LIN {X 0,Y 332.118,Z 721.88,A -85,B 0,C 180,E1 -12190.22,E2 -12190.22} C_VEL
LIN {X 0,Y 333.86,Z 711.932,A -85,B 0,C 180,E1 -12192.438,E2 -12192.438} C_VEL
LIN {X 0,Y 335.853,Z 699.998,A -85,B 0,C 180,E1 -12194.532,E2 -12194.532} C_VEL
LIN {X 0,Y 337.763,Z 687.766,A -85,B 0,C 180,E1 -12196.241,E2 -12196.241} C_VEL
LIN {X 0,Y 339.691,Z 673.523,A -85,B 0,C 180,E1 -12197.797,E2 -12197.797} C_VEL
LIN {X 0,Y 341.315,Z 659.406,A -85,B 0,C 180,E1 -12198.989,E2 -12198.989} C_VEL
LIN {X 0,Y 342.676,Z 643.422,A -85,B 0,C 180,E1 -12199.976,E2 -12199.976} C_VEL
LIN {X 0,Y 343.599,Z 627.214,A -85,B 0,C 180,E1 -12200.656,E2 -12200.656} C_VEL
LIN {X 0,Y 345.215,Z 570.987,A -85,B 0,C 180,E1 -12201.908,E2 -12201.908} C_VEL
LIN {X 0,Y 347.175,Z 499.948,A -85,B 0,C 180,E1 -12203.441,E2 -12203.441} C_VEL
LIN {X 0,Y 345.23,Z 482.09,A -85,B 0,C 180,E1 -12204.102,E2 -12204.102} C_VEL
LIN {X 0,Y 348.72,Z 438.304,A -85,B 0,C 180,E1 -12208.447,E2 -12208.447} C_VEL
LIN {X 0,Y 351.971,Z 398.894,A -85,B 0,C 180,E1 -12212.333,E2 -12212.333} C_VEL
LIN {X 0,Y 355.002,Z 360.835,A -85,B 0,C 180,E1 -12216.072,E2 -12216.072} C_VEL
LIN {X 0,Y 355.314,Z 355.414,A -85,B 0,C 180,E1 -12216.623,E2 -12216.623} C_VEL
LIN {X 0,Y 350.277,Z 339.623,A -85,B 0,C 180,E1 -12219.095,E2 -12219.095} C_VEL
LIN {X 0,Y 344.773,Z 325.615,A -85,B 0,C 180,E1 -12221.572,E2 -12221.572} C_VEL
LIN {X 0,Y 338.807,Z 312.634,A -85,B 0,C 180,E1 -12224.158,E2 -12224.158} C_VEL
LIN {X 0,Y 334.604,Z 304.41,A -85,B 0,C 180,E1 -12225.992,E2 -12225.992} C_VEL
LIN {X 0,Y 332,Z 299.711,A -85,B 0,C 180,E1 -12227.122,E2 -12227.122} C_VEL
LIN {X 0,Y 330.195,Z 296.3,A -85,B 0,C 180,E1 -12227.959,E2 -12227.959} C_VEL
LIN {X 0,Y 330.046,Z 295.41,A -85,B 0,C 180,E1 -12228.363,E2 -12228.363} C_VEL
LIN {X 0,Y 330.062,Z 295.372,A -85,B 0,C 180,E1 -12232.69,E2 -12232.69} C_VEL
LIN {X 0,Y 330.038,Z 295.376,A -85,B 0,C 180,E1 -12237.047,E2 -12237.047} C_VEL
LIN {X 0,Y 330.027,Z 295.369,A -85,B 0,C 180,E1 -12241.388,E2 -12241.388} C_VEL
LIN {X 0,Y 330.023,Z 295.376,A -85,B 0,C 180,E1 -12245.737,E2 -12245.737} C_VEL
LIN {X 0,Y 330.026,Z 295.368,A -85,B 0,C 180,E1 -12250.12,E2 -12250.12} C_VEL
LIN {X 0,Y 330.038,Z 295.376,A -85,B 0,C 180,E1 -12254.383,E2 -12254.383} C_VEL
LIN {X 0,Y 330.048,Z 295.365,A -85,B 0,C 180,E1 -12258.73,E2 -12258.73} C_VEL
LIN {X 0,Y 330.059,Z 295.37,A -85,B 0,C 180,E1 -12263.003,E2 -12263.003} C_VEL
LIN {X 0,Y 330.042,Z 295.369,A -85,B 0,C 180,E1 -12267.427,E2 -12267.427} C_VEL
LIN {X 0,Y 330.036,Z 295.371,A -85,B 0,C 180,E1 -12271.651,E2 -12271.651} C_VEL
LIN {X 0,Y 330.069,Z 295.642,A -85,B 0,C 180,E1 -12274.026,E2 -12274.026} C_VEL
LIN {X 0,Y 331.671,Z 299.336,A -85,B 0,C 180,E1 -12274.943,E2 -12274.943} C_VEL
LIN {X 0,Y 339.158,Z 316.344,A -85,B 0,C 180,E1 -12278.681,E2 -12278.681} C_VEL
LIN {X 0,Y 341.505,Z 321.378,A -85,B 0,C 180,E1 -12279.662,E2 -12279.662} C_VEL
LIN {X 0,Y 357.451,Z 348.34,A -85,B 0,C 180,E1 -12282.794,E2 -12282.794} C_VEL
LIN {X 0,Y 370.048,Z 371.248,A -85,B 0,C 180,E1 -12285.081,E2 -12285.081} C_VEL
LIN {X 0,Y 357.996,Z 576.955,A -85,B 0,C 180,E1 -12290.185,E2 -12290.185} C_VEL
LIN {X 0,Y 355.992,Z 598.538,A -85,B 0,C 180,E1 -12291.003,E2 -12291.003} C_VEL
LIN {X 0,Y 353.569,Z 618.824,A -85,B 0,C 180,E1 -12292.056,E2 -12292.056} C_VEL
LIN {X 0,Y 350.696,Z 639.126,A -85,B 0,C 180,E1 -12293.428,E2 -12293.428} C_VEL
LIN {X 0,Y 347.572,Z 658.567,A -85,B 0,C 180,E1 -12295.081,E2 -12295.081} C_VEL
LIN {X 0,Y 344.166,Z 677.781,A -85,B 0,C 180,E1 -12297.096,E2 -12297.096} C_VEL
LIN {X 0,Y 340.909,Z 695.134,A -85,B 0,C 180,E1 -12299.317,E2 -12299.317} C_VEL
LIN {X 0,Y 337.768,Z 711.391,A -85,B 0,C 180,E1 -12301.829,E2 -12301.829} C_VEL
LIN {X 0,Y 334.968,Z 725.97,A -85,B 0,C 180,E1 -12304.546,E2 -12304.546} C_VEL
LIN {X 0,Y 332.525,Z 739.34,A -85,B 0,C 180,E1 -12307.553,E2 -12307.553} C_VEL
LIN {X 0,Y 330.674,Z 750.572,A -85,B 0,C 180,E1 -12310.628,E2 -12310.628} C_VEL
LIN {X 0,Y 329.371,Z 759.964,A -85,B 0,C 180,E1 -12313.785,E2 -12313.785} C_VEL
LIN {X 0,Y 328.56,Z 767.582,A -85,B 0,C 180,E1 -12316.988,E2 -12316.988} C_VEL
LIN {X 0,Y 328.163,Z 773.719,A -85,B 0,C 180,E1 -12320.355,E2 -12320.355} C_VEL
LIN {X 0,Y 328.074,Z 777.864,A -85,B 0,C 180,E1 -12323.527,E2 -12323.527} C_VEL
LIN {X 0,Y 328.085,Z 780.383,A -85,B 0,C 180,E1 -12326.682,E2 -12326.682} C_VEL
LIN {X 0,Y 328.118,Z 781.355,A -85,B 0,C 180,E1 -12329.827,E2 -12329.827} C_VEL
LIN {X 0,Y 328.075,Z 780.859,A -85,B 0,C 180,E1 -12332.972,E2 -12332.972} C_VEL
LIN {X 0,Y 328.045,Z 778.829,A -85,B 0,C 180,E1 -12336.126,E2 -12336.126} C_VEL
LIN {X 0,Y 328.116,Z 775.251,A -85,B 0,C 180,E1 -12339.296,E2 -12339.296} C_VEL
LIN {X 0,Y 328.493,Z 769.816,A -85,B 0,C 180,E1 -12342.661,E2 -12342.661} C_VEL
LIN {X 0,Y 329.298,Z 763.002,A -85,B 0,C 180,E1 -12345.861,E2 -12345.861} C_VEL
LIN {X 0,Y 330.734,Z 753.863,A -85,B 0,C 180,E1 -12349.242,E2 -12349.242} C_VEL
LIN {X 0,Y 332.904,Z 742.52,A -85,B 0,C 180,E1 -12352.611,E2 -12352.611} C_VEL
LIN {X 0,Y 335.725,Z 729.474,A -85,B 0,C 180,E1 -12355.775,E2 -12355.775} C_VEL
LIN {X 0,Y 339.122,Z 714.749,A -85,B 0,C 180,E1 -12358.725,E2 -12358.725} C_VEL
LIN {X 0,Y 343.041,Z 698.333,A -85,B 0,C 180,E1 -12361.45,E2 -12361.45} C_VEL
LIN {X 0,Y 347.215,Z 680.841,A -85,B 0,C 180,E1 -12363.865,E2 -12363.865} C_VEL
LIN {X 0,Y 351.726,Z 661.714,A -85,B 0,C 180,E1 -12366.048,E2 -12366.048} C_VEL
LIN {X 0,Y 356.386,Z 641.227,A -85,B 0,C 180,E1 -12367.968,E2 -12367.968} C_VEL
LIN {X 0,Y 360.995,Z 620.134,A -85,B 0,C 180,E1 -12369.573,E2 -12369.573} C_VEL
LIN {X 0,Y 365.603,Z 597.763,A -85,B 0,C 180,E1 -12370.92,E2 -12370.92} C_VEL
LIN {X 0,Y 370.108,Z 573.956,A -85,B 0,C 180,E1 -12372.002,E2 -12372.002} C_VEL
LIN {X 0,Y 380.25,Z 515.563,A -85,B 0,C 180,E1 -12374.095,E2 -12374.095} C_VEL
LIN {X 0,Y 391.481,Z 464.537,A -85,B 0,C 180,E1 -12375.931,E2 -12375.931} C_VEL
LIN {X 0,Y 399.695,Z 432.421,A -85,B 0,C 180,E1 -12377.075,E2 -12377.075} C_VEL
LIN {X 0,Y 383.918,Z 497.009,A -85,B 0,C 180,E1 -12379.426,E2 -12379.426} C_VEL
LIN {X 0,Y 372.15,Z 555.463,A -85,B 0,C 180,E1 -12381.651,E2 -12381.651} C_VEL
LIN {X 0,Y 367.645,Z 579.27,A -85,B 0,C 180,E1 -12382.665,E2 -12382.665} C_VEL
LIN {X 0,Y 363.116,Z 600.549,A -85,B 0,C 180,E1 -12383.896,E2 -12383.896} C_VEL
LIN {X 0,Y 358.234,Z 621.939,A -85,B 0,C 180,E1 -12385.488,E2 -12385.488} C_VEL
LIN {X 0,Y 353.563,Z 641.476,A -85,B 0,C 180,E1 -12387.308,E2 -12387.308} C_VEL
LIN {X 0,Y 349.098,Z 659.317,A -85,B 0,C 180,E1 -12389.349,E2 -12389.349} C_VEL
LIN {X 0,Y 344.901,Z 675.585,A -85,B 0,C 180,E1 -12391.613,E2 -12391.613} C_VEL
LIN {X 0,Y 341.034,Z 690.337,A -85,B 0,C 180,E1 -12394.098,E2 -12394.098} C_VEL
LIN {X 0,Y 337.575,Z 703.545,A -85,B 0,C 180,E1 -12396.801,E2 -12396.801} C_VEL
LIN {X 0,Y 334.599,Z 715.171,A -85,B 0,C 180,E1 -12399.719,E2 -12399.719} C_VEL
LIN {X 0,Y 332.292,Z 724.649,A -85,B 0,C 180,E1 -12402.67,E2 -12402.67} C_VEL
LIN {X 0,Y 330.597,Z 732.231,A -85,B 0,C 180,E1 -12405.641,E2 -12405.641} C_VEL
LIN {X 0,Y 329.386,Z 738.403,A -85,B 0,C 180,E1 -12408.798,E2 -12408.798} C_VEL
LIN {X 0,Y 328.658,Z 742.803,A -85,B 0,C 180,E1 -12411.956,E2 -12411.956} C_VEL
LIN {X 0,Y 328.278,Z 745.629,A -85,B 0,C 180,E1 -12415.284,E2 -12415.284} C_VEL
LIN {X 0,Y 328.142,Z 746.633,A -85,B 0,C 180,E1 -12418.429,E2 -12418.429} C_VEL
LIN {X 0,Y 328.103,Z 746.012,A -85,B 0,C 180,E1 -12421.572,E2 -12421.572} C_VEL
LIN {X 0,Y 328.151,Z 743.758,A -85,B 0,C 180,E1 -12424.72,E2 -12424.72} C_VEL
LIN {X 0,Y 328.372,Z 739.807,A -85,B 0,C 180,E1 -12427.876,E2 -12427.876} C_VEL
LIN {X 0,Y 328.849,Z 734.444,A -85,B 0,C 180,E1 -12430.867,E2 -12430.867} C_VEL
LIN {X 0,Y 329.72,Z 727.043,A -85,B 0,C 180,E1 -12433.975,E2 -12433.975} C_VEL
LIN {X 0,Y 330.982,Z 718.343,A -85,B 0,C 180,E1 -12436.859,E2 -12436.859} C_VEL
LIN {X 0,Y 332.702,Z 707.869,A -85,B 0,C 180,E1 -12439.67,E2 -12439.67} C_VEL
LIN {X 0,Y 334.795,Z 695.999,A -85,B 0,C 180,E1 -12442.29,E2 -12442.29} C_VEL
LIN {X 0,Y 337.291,Z 682.225,A -85,B 0,C 180,E1 -12444.801,E2 -12444.801} C_VEL
LIN {X 0,Y 339.946,Z 667.484,A -85,B 0,C 180,E1 -12447.028,E2 -12447.028} C_VEL
LIN {X 0,Y 342.754,Z 651.22,A -85,B 0,C 180,E1 -12449.059,E2 -12449.059} C_VEL
LIN {X 0,Y 345.512,Z 634.102,A -85,B 0,C 180,E1 -12450.812,E2 -12450.812} C_VEL
LIN {X 0,Y 348.253,Z 615.141,A -85,B 0,C 180,E1 -12452.376,E2 -12452.376} C_VEL
LIN {X 0,Y 350.723,Z 595.391,A -85,B 0,C 180,E1 -12453.647,E2 -12453.647} C_VEL
LIN {X 0,Y 352.768,Z 575.246,A -85,B 0,C 180,E1 -12454.618,E2 -12454.618} C_VEL
LIN {X 0,Y 354.34,Z 554.645,A -85,B 0,C 180,E1 -12455.306,E2 -12455.306} C_VEL
LIN {X 0,Y 364.432,Z 383.187,A -85,B 0,C 180,E1 -12459.733,E2 -12459.733} C_VEL
LIN {X 0,Y 362.119,Z 366.133,A -85,B 0,C 180,E1 -12460.564,E2 -12460.564} C_VEL
LIN {X 0,Y 348.934,Z 341.464,A -85,B 0,C 180,E1 -12463.054,E2 -12463.054} C_VEL
LIN {X 0,Y 347.117,Z 337.74,A -85,B 0,C 180,E1 -12463.507,E2 -12463.507} C_VEL
LIN {X 0,Y 339.998,Z 319.459,A -85,B 0,C 180,E1 -12467.208,E2 -12467.208} C_VEL
LIN {X 0,Y 333.092,Z 302.809,A -85,B 0,C 180,E1 -12470.921,E2 -12470.921} C_VEL
LIN {X 0,Y 330.076,Z 295.57,A -85,B 0,C 180,E1 -12472.715,E2 -12472.715} C_VEL
LIN {X 0,Y 330.043,Z 295.371,A -85,B 0,C 180,E1 -12477.054,E2 -12477.054} C_VEL
LIN {X 0,Y 330.044,Z 295.349,A -85,B 0,C 180,E1 -12481.469,E2 -12481.469} C_VEL
LIN {X 0,Y 330.072,Z 295.561,A -85,B 0,C 180,E1 -12483.653,E2 -12483.653} C_VEL
LIN {X 0,Y 330.669,Z 297.596,A -85,B 0,C 180,E1 -12484.103,E2 -12484.103} C_VEL
LIN {X 0,Y 332.502,Z 301.305,A -85,B 0,C 180,E1 -12484.843,E2 -12484.843} C_VEL
LIN {X 0,Y 338.631,Z 314.413,A -85,B 0,C 180,E1 -12487.335,E2 -12487.335} C_VEL
LIN {X 0,Y 346.07,Z 332.865,A -85,B 0,C 180,E1 -12490.496,E2 -12490.496} C_VEL
LIN {X 0,Y 352.203,Z 350.651,A -85,B 0,C 180,E1 -12493.251,E2 -12493.251} C_VEL
LIN {X 0,Y 353.624,Z 356.013,A -85,B 0,C 180,E1 -12494.018,E2 -12494.018} C_VEL
LIN {X 0,Y 350.25,Z 397.698,A -85,B 0,C 180,E1 -12498.188,E2 -12498.188} C_VEL
LIN {X 0,Y 346.855,Z 438.589,A -85,B 0,C 180,E1 -12502.295,E2 -12502.295} C_VEL
LIN {X 0,Y 343.61,Z 481.813,A -85,B 0,C 180,E1 -12506.589,E2 -12506.589} C_VEL
LIN {X 0,Y 345.615,Z 502.467,A -85,B 0,C 180,E1 -12507.247,E2 -12507.247} C_VEL
LIN {X 0,Y 344.007,Z 560.903,A -85,B 0,C 180,E1 -12508.478,E2 -12508.478} C_VEL
LIN {X 0,Y 342.903,Z 568.569,A -85,B 0,C 180,E1 -12508.569,E2 -12508.569} C_VEL
LIN {X 0,Y 336.694,Z 588.888,A -85,B 0,C 180,E1 -12508.554,E2 -12508.554} C_VEL
LIN {X 0,Y 335.813,Z 595.472,A -85,B 0,C 180,E1 -12508.639,E2 -12508.639} C_VEL
LIN {X 0,Y 334.887,Z 627.398,A -85,B 0,C 180,E1 -12509.389,E2 -12509.389} C_VEL
LIN {X 0,Y 333.893,Z 644.369,A -85,B 0,C 180,E1 -12510.132,E2 -12510.132} C_VEL
LIN {X 0,Y 332.58,Z 659.659,A -85,B 0,C 180,E1 -12511.118,E2 -12511.118} C_VEL
LIN {X 0,Y 330.794,Z 675.437,A -85,B 0,C 180,E1 -12512.51,E2 -12512.51} C_VEL
LIN {X 0,Y 328.935,Z 689.154,A -85,B 0,C 180,E1 -12514.094,E2 -12514.094} C_VEL
LIN {X 0,Y 326.922,Z 702.47,A -85,B 0,C 180,E1 -12516.055,E2 -12516.055} C_VEL
LIN {X 0,Y 325.117,Z 713.568,A -85,B 0,C 180,E1 -12518.131,E2 -12518.131} C_VEL
LIN {X 0,Y 323.428,Z 723.844,A -85,B 0,C 180,E1 -12520.551,E2 -12520.551} C_VEL
LIN {X 0,Y 322.094,Z 732.194,A -85,B 0,C 180,E1 -12523.095,E2 -12523.095} C_VEL
LIN {X 0,Y 321.1,Z 739.181,A -85,B 0,C 180,E1 -12525.901,E2 -12525.901} C_VEL
LIN {X 0,Y 320.51,Z 744.121,A -85,B 0,C 180,E1 -12528.74,E2 -12528.74} C_VEL
LIN {X 0,Y 320.237,Z 747.308,A -85,B 0,C 180,E1 -12531.616,E2 -12531.616} C_VEL
LIN {X 0,Y 320.153,Z 748.689,A -85,B 0,C 180,E1 -12534.54,E2 -12534.54} C_VEL
LIN {X 0,Y 320.208,Z 748.308,A -85,B 0,C 180,E1 -12537.525,E2 -12537.525} C_VEL
LIN {X 0,Y 320.437,Z 746.187,A -85,B 0,C 180,E1 -12540.361,E2 -12540.361} C_VEL
LIN {X 0,Y 320.956,Z 742.246,A -85,B 0,C 180,E1 -12543.247,E2 -12543.247} C_VEL
LIN {X 0,Y 321.823,Z 736.738,A -85,B 0,C 180,E1 -12545.955,E2 -12545.955} C_VEL
LIN {X 0,Y 323.216,Z 728.85,A -85,B 0,C 180,E1 -12548.779,E2 -12548.779} C_VEL
LIN {X 0,Y 324.847,Z 719.976,A -85,B 0,C 180,E1 -12551.196,E2 -12551.196} C_VEL
LIN {X 0,Y 326.856,Z 709.046,A -85,B 0,C 180,E1 -12553.531,E2 -12553.531} C_VEL
LIN {X 0,Y 328.852,Z 697.514,A -85,B 0,C 180,E1 -12555.475,E2 -12555.475} C_VEL
LIN {X 0,Y 331.034,Z 683.779,A -85,B 0,C 180,E1 -12557.306,E2 -12557.306} C_VEL
LIN {X 0,Y 332.952,Z 669.65,A -85,B 0,C 180,E1 -12558.762,E2 -12558.762} C_VEL
LIN {X 0,Y 334.649,Z 654.366,A -85,B 0,C 180,E1 -12559.958,E2 -12559.958} C_VEL
LIN {X 0,Y 335.907,Z 638.471,A -85,B 0,C 180,E1 -12560.845,E2 -12560.845} C_VEL
LIN {X 0,Y 336.731,Z 621.67,A -85,B 0,C 180,E1 -12561.447,E2 -12561.447} C_VEL
LIN {X 0,Y 340.273,Z 500.964,A -85,B 0,C 180,E1 -12564.097,E2 -12564.097} C_VEL
LIN {X 0,Y 338.291,Z 482.445,A -85,B 0,C 180,E1 -12564.805,E2 -12564.805} C_VEL
LIN {X 0,Y 342.014,Z 438.182,A -85,B 0,C 180,E1 -12569.255,E2 -12569.255} C_VEL
LIN {X 0,Y 345.643,Z 397.177,A -85,B 0,C 180,E1 -12573.357,E2 -12573.357} C_VEL
LIN {X 0,Y 348.845,Z 358.991,A -85,B 0,C 180,E1 -12577.146,E2 -12577.146} C_VEL
LIN {X 0,Y 344.084,Z 343.766,A -85,B 0,C 180,E1 -12579.591,E2 -12579.591} C_VEL
LIN {X 0,Y 338.376,Z 328.993,A -85,B 0,C 180,E1 -12582.28,E2 -12582.28} C_VEL
LIN {X 0,Y 331.614,Z 314.432,A -85,B 0,C 180,E1 -12585.328,E2 -12585.328} C_VEL
LIN {X 0,Y 326.919,Z 305.633,A -85,B 0,C 180,E1 -12587.458,E2 -12587.458} C_VEL
LIN {X 0,Y 324.243,Z 300.882,A -85,B 0,C 180,E1 -12588.684,E2 -12588.684} C_VEL
LIN {X 0,Y 322.535,Z 298.193,A -85,B 0,C 180,E1 -12589.461,E2 -12589.461} C_VEL
LIN {X 0,Y 322.105,Z 296.499,A -85,B 0,C 180,E1 -12589.989,E2 -12589.989} C_VEL
LIN {X 0,Y 322.099,Z 296.361,A -85,B 0,C 180,E1 -12594.298,E2 -12594.298} C_VEL
LIN {X 0,Y 322.113,Z 296.356,A -85,B 0,C 180,E1 -12598.754,E2 -12598.754} C_VEL
LIN {X 0,Y 322.102,Z 296.36,A -85,B 0,C 180,E1 -12603.024,E2 -12603.024} C_VEL
LIN {X 0,Y 322.1,Z 296.357,A -85,B 0,C 180,E1 -12607.311,E2 -12607.311} C_VEL
LIN {X 0,Y 322.087,Z 296.364,A -85,B 0,C 180,E1 -12611.64,E2 -12611.64} C_VEL
LIN {X 0,Y 322.086,Z 296.356,A -85,B 0,C 180,E1 -12616.038,E2 -12616.038} C_VEL
LIN {X 0,Y 322.097,Z 296.365,A -85,B 0,C 180,E1 -12620.376,E2 -12620.376} C_VEL
LIN {X 0,Y 322.103,Z 296.358,A -85,B 0,C 180,E1 -12624.579,E2 -12624.579} C_VEL
LIN {X 0,Y 322.126,Z 296.358,A -85,B 0,C 180,E1 -12628.96,E2 -12628.96} C_VEL
LIN {X 0,Y 322.141,Z 296.599,A -85,B 0,C 180,E1 -12632.745,E2 -12632.745} C_VEL
LIN {X 0,Y 323.437,Z 299.898,A -85,B 0,C 180,E1 -12633.597,E2 -12633.597} C_VEL
LIN {X 0,Y 329.487,Z 313.282,A -85,B 0,C 180,E1 -12636.713,E2 -12636.713} C_VEL
LIN {X 0,Y 333.208,Z 321.551,A -85,B 0,C 180,E1 -12638.451,E2 -12638.451} C_VEL
LIN {X 0,Y 347.955,Z 346.12,A -85,B 0,C 180,E1 -12641.479,E2 -12641.479} C_VEL
LIN {X 0,Y 363.468,Z 373.851,A -85,B 0,C 180,E1 -12644.396,E2 -12644.396} C_VEL
LIN {X 0,Y 351.024,Z 576.718,A -85,B 0,C 180,E1 -12649.549,E2 -12649.549} C_VEL
LIN {X 0,Y 349.008,Z 597.716,A -85,B 0,C 180,E1 -12650.354,E2 -12650.354} C_VEL
LIN {X 0,Y 346.442,Z 618.576,A -85,B 0,C 180,E1 -12651.455,E2 -12651.455} C_VEL
LIN {X 0,Y 343.484,Z 638.791,A -85,B 0,C 180,E1 -12652.845,E2 -12652.845} C_VEL
LIN {X 0,Y 340.27,Z 658.146,A -85,B 0,C 180,E1 -12654.518,E2 -12654.518} C_VEL
LIN {X 0,Y 336.815,Z 677.039,A -85,B 0,C 180,E1 -12656.529,E2 -12656.529} C_VEL
LIN {X 0,Y 333.395,Z 694.677,A -85,B 0,C 180,E1 -12658.822,E2 -12658.822} C_VEL
LIN {X 0,Y 330.106,Z 711.106,A -85,B 0,C 180,E1 -12661.411,E2 -12661.411} C_VEL
LIN {X 0,Y 327.119,Z 726.145,A -85,B 0,C 180,E1 -12664.279,E2 -12664.279} C_VEL
LIN {X 0,Y 324.605,Z 739.455,A -85,B 0,C 180,E1 -12667.357,E2 -12667.357} C_VEL
LIN {X 0,Y 322.639,Z 751.062,A -85,B 0,C 180,E1 -12670.637,E2 -12670.637} C_VEL
LIN {X 0,Y 321.313,Z 760.445,A -85,B 0,C 180,E1 -12673.924,E2 -12673.924} C_VEL
LIN {X 0,Y 320.522,Z 767.872,A -85,B 0,C 180,E1 -12677.206,E2 -12677.206} C_VEL
LIN {X 0,Y 320.163,Z 773.545,A -85,B 0,C 180,E1 -12680.475,E2 -12680.475} C_VEL
LIN {X 0,Y 320.084,Z 777.59,A -85,B 0,C 180,E1 -12683.725,E2 -12683.725} C_VEL
LIN {X 0,Y 320.103,Z 780.047,A -85,B 0,C 180,E1 -12686.958,E2 -12686.958} C_VEL
LIN {X 0,Y 320.131,Z 780.898,A -85,B 0,C 180,E1 -12690.181,E2 -12690.181} C_VEL
LIN {X 0,Y 320.076,Z 780.269,A -85,B 0,C 180,E1 -12693.405,E2 -12693.405} C_VEL
LIN {X 0,Y 320.049,Z 778.155,A -85,B 0,C 180,E1 -12696.64,E2 -12696.64} C_VEL
LIN {X 0,Y 320.158,Z 774.434,A -85,B 0,C 180,E1 -12699.892,E2 -12699.892} C_VEL
LIN {X 0,Y 320.623,Z 768.833,A -85,B 0,C 180,E1 -12703.354,E2 -12703.354} C_VEL
LIN {X 0,Y 321.634,Z 761.444,A -85,B 0,C 180,E1 -12706.806,E2 -12706.806} C_VEL
LIN {X 0,Y 323.208,Z 752.634,A -85,B 0,C 180,E1 -12710.085,E2 -12710.085} C_VEL
LIN {X 0,Y 325.492,Z 741.846,A -85,B 0,C 180,E1 -12713.347,E2 -12713.347} C_VEL
LIN {X 0,Y 328.572,Z 728.823,A -85,B 0,C 180,E1 -12716.574,E2 -12716.574} C_VEL
LIN {X 0,Y 332.275,Z 714.126,A -85,B 0,C 180,E1 -12719.584,E2 -12719.584} C_VEL
LIN {X 0,Y 336.498,Z 697.928,A -85,B 0,C 180,E1 -12722.335,E2 -12722.335} C_VEL
LIN {X 0,Y 341.157,Z 680.064,A -85,B 0,C 180,E1 -12724.857,E2 -12724.857} C_VEL
LIN {X 0,Y 346.019,Z 661.29,A -85,B 0,C 180,E1 -12727.05,E2 -12727.05} C_VEL
LIN {X 0,Y 351.14,Z 641.007,A -85,B 0,C 180,E1 -12728.999,E2 -12728.999} C_VEL
LIN {X 0,Y 356.482,Z 619.129,A -85,B 0,C 180,E1 -12730.703,E2 -12730.703} C_VEL
LIN {X 0,Y 361.756,Z 596.519,A -85,B 0,C 180,E1 -12732.088,E2 -12732.088} C_VEL
LIN {X 0,Y 366.888,Z 572.676,A -85,B 0,C 180,E1 -12733.188,E2 -12733.188} C_VEL
LIN {X 0,Y 377.868,Z 517.801,A -85,B 0,C 180,E1 -12735.207,E2 -12735.207} C_VEL
LIN {X 0,Y 390.643,Z 466.175,A -85,B 0,C 180,E1 -12737.08,E2 -12737.08} C_VEL
LIN {X 0,Y 375.431,Z 527.422,A -85,B 0,C 180,E1 -12739.384,E2 -12739.384} C_VEL
LIN {X 0,Y 365.285,Z 574.697,A -85,B 0,C 180,E1 -12741.285,E2 -12741.285} C_VEL
LIN {X 0,Y 360.226,Z 596.098,A -85,B 0,C 180,E1 -12742.465,E2 -12742.465} C_VEL
LIN {X 0,Y 355.032,Z 616.708,A -85,B 0,C 180,E1 -12743.943,E2 -12743.943} C_VEL
LIN {X 0,Y 349.752,Z 636.453,A -85,B 0,C 180,E1 -12745.725,E2 -12745.725} C_VEL
LIN {X 0,Y 344.549,Z 655.366,A -85,B 0,C 180,E1 -12747.826,E2 -12747.826} C_VEL
LIN {X 0,Y 339.7,Z 672.619,A -85,B 0,C 180,E1 -12750.171,E2 -12750.171} C_VEL
LIN {X 0,Y 335.344,Z 687.875,A -85,B 0,C 180,E1 -12752.69,E2 -12752.69} C_VEL
LIN {X 0,Y 331.458,Z 701.373,A -85,B 0,C 180,E1 -12755.4,E2 -12755.4} C_VEL
LIN {X 0,Y 328.046,Z 713.374,A -85,B 0,C 180,E1 -12758.359,E2 -12758.359} C_VEL
LIN {X 0,Y 325.36,Z 723.236,A -85,B 0,C 180,E1 -12761.362,E2 -12761.362} C_VEL
LIN {X 0,Y 323.337,Z 731.206,A -85,B 0,C 180,E1 -12764.394,E2 -12764.394} C_VEL
LIN {X 0,Y 321.844,Z 737.757,A -85,B 0,C 180,E1 -12767.623,E2 -12767.623} C_VEL
LIN {X 0,Y 320.915,Z 742.528,A -85,B 0,C 180,E1 -12770.858,E2 -12770.858} C_VEL
LIN {X 0,Y 320.397,Z 745.718,A -85,B 0,C 180,E1 -12774.269,E2 -12774.269} C_VEL
LIN {X 0,Y 320.185,Z 747.083,A -85,B 0,C 180,E1 -12777.495,E2 -12777.495} C_VEL
LIN {X 0,Y 320.124,Z 746.801,A -85,B 0,C 180,E1 -12780.716,E2 -12780.716} C_VEL
LIN {X 0,Y 320.137,Z 744.879,A -85,B 0,C 180,E1 -12783.941,E2 -12783.941} C_VEL
LIN {X 0,Y 320.308,Z 741.283,A -85,B 0,C 180,E1 -12787.173,E2 -12787.173} C_VEL
LIN {X 0,Y 320.76,Z 735.921,A -85,B 0,C 180,E1 -12790.417,E2 -12790.417} C_VEL
LIN {X 0,Y 321.553,Z 729.098,A -85,B 0,C 180,E1 -12793.487,E2 -12793.487} C_VEL
LIN {X 0,Y 322.818,Z 720.405,A -85,B 0,C 180,E1 -12796.557,E2 -12796.557} C_VEL
LIN {X 0,Y 324.538,Z 710.111,A -85,B 0,C 180,E1 -12799.479,E2 -12799.479} C_VEL
LIN {X 0,Y 326.746,Z 697.947,A -85,B 0,C 180,E1 -12802.3,E2 -12802.3} C_VEL
LIN {X 0,Y 329.37,Z 683.992,A -85,B 0,C 180,E1 -12804.959,E2 -12804.959} C_VEL
LIN {X 0,Y 332.191,Z 668.881,A -85,B 0,C 180,E1 -12807.324,E2 -12807.324} C_VEL
LIN {X 0,Y 335.198,Z 652.054,A -85,B 0,C 180,E1 -12809.485,E2 -12809.485} C_VEL
LIN {X 0,Y 337.999,Z 635.314,A -85,B 0,C 180,E1 -12811.248,E2 -12811.248} C_VEL
LIN {X 0,Y 340.71,Z 617.38,A -85,B 0,C 180,E1 -12812.783,E2 -12812.783} C_VEL
LIN {X 0,Y 343.225,Z 598.27,A -85,B 0,C 180,E1 -12814.075,E2 -12814.075} C_VEL
LIN {X 0,Y 345.44,Z 577.827,A -85,B 0,C 180,E1 -12815.12,E2 -12815.12} C_VEL
LIN {X 0,Y 347.173,Z 556.743,A -85,B 0,C 180,E1 -12815.871,E2 -12815.871} C_VEL
LIN {X 0,Y 357.874,Z 384.361,A -85,B 0,C 180,E1 -12820.449,E2 -12820.449} C_VEL
LIN {X 0,Y 355.884,Z 369.657,A -85,B 0,C 180,E1 -12821.182,E2 -12821.182} C_VEL
LIN {X 0,Y 341.429,Z 342.54,A -85,B 0,C 180,E1 -12824.001,E2 -12824.001} C_VEL
LIN {X 0,Y 338.884,Z 337.675,A -85,B 0,C 180,E1 -12824.605,E2 -12824.605} C_VEL
LIN {X 0,Y 331.893,Z 319.885,A -85,B 0,C 180,E1 -12828.343,E2 -12828.343} C_VEL
LIN {X 0,Y 325.215,Z 303.882,A -85,B 0,C 180,E1 -12832.054,E2 -12832.054} C_VEL
LIN {X 0,Y 322.135,Z 296.54,A -85,B 0,C 180,E1 -12833.931,E2 -12833.931} C_VEL
LIN {X 0,Y 322.115,Z 296.361,A -85,B 0,C 180,E1 -12838.358,E2 -12838.358} C_VEL
LIN {X 0,Y 322.138,Z 296.597,A -85,B 0,C 180,E1 -12842.452,E2 -12842.452} C_VEL
LIN {X 0,Y 323.046,Z 299.275,A -85,B 0,C 180,E1 -12843.05,E2 -12843.05} C_VEL
LIN {X 0,Y 324.547,Z 302.103,A -85,B 0,C 180,E1 -12843.662,E2 -12843.662} C_VEL
LIN {X 0,Y 331.128,Z 316.025,A -85,B 0,C 180,E1 -12846.413,E2 -12846.413} C_VEL
LIN {X 0,Y 338.332,Z 333.564,A -85,B 0,C 180,E1 -12849.526,E2 -12849.526} C_VEL
LIN {X 0,Y 344.673,Z 351.685,A -85,B 0,C 180,E1 -12852.439,E2 -12852.439} C_VEL
LIN {X 0,Y 346.739,Z 358.83,A -85,B 0,C 180,E1 -12853.497,E2 -12853.497} C_VEL
LIN {X 0,Y 343.159,Z 400.438,A -85,B 0,C 180,E1 -12857.718,E2 -12857.718} C_VEL
LIN {X 0,Y 339.592,Z 442.338,A -85,B 0,C 180,E1 -12861.959,E2 -12861.959} C_VEL
LIN {X 0,Y 336.435,Z 482.085,A -85,B 0,C 180,E1 -12865.961,E2 -12865.961} C_VEL
LIN {X 0,Y 338.461,Z 503.376,A -85,B 0,C 180,E1 -12866.656,E2 -12866.656} C_VEL
LIN {X 0,Y 335.813,Z 595.472,A -85,B 0,C 180,E1 -12868.639,E2 -12868.639} C_VEL
LIN {X 0,Y 334.693,Z 603.149,A -85,B 0,C 180,E1 -12868.723,E2 -12868.723} C_VEL
LIN {X 0,Y 328.705,Z 622.369,A -85,B 0,C 180,E1 -12868.727,E2 -12868.727} C_VEL
LIN {X 0,Y 327.484,Z 629.952,A -85,B 0,C 180,E1 -12868.905,E2 -12868.905} C_VEL
LIN {X 0,Y 326.471,Z 645.96,A -85,B 0,C 180,E1 -12869.647,E2 -12869.647} C_VEL
LIN {X 0,Y 325.031,Z 661.476,A -85,B 0,C 180,E1 -12870.703,E2 -12870.703} C_VEL
LIN {X 0,Y 323.294,Z 676.092,A -85,B 0,C 180,E1 -12872.036,E2 -12872.036} C_VEL
LIN {X 0,Y 321.355,Z 689.746,A -85,B 0,C 180,E1 -12873.655,E2 -12873.655} C_VEL
LIN {X 0,Y 319.343,Z 702.477,A -85,B 0,C 180,E1 -12875.568,E2 -12875.568} C_VEL
LIN {X 0,Y 317.522,Z 713.237,A -85,B 0,C 180,E1 -12877.598,E2 -12877.598} C_VEL
LIN {X 0,Y 315.747,Z 723.463,A -85,B 0,C 180,E1 -12880.028,E2 -12880.028} C_VEL
LIN {X 0,Y 314.38,Z 731.614,A -85,B 0,C 180,E1 -12882.488,E2 -12882.488} C_VEL
LIN {X 0,Y 313.266,Z 738.806,A -85,B 0,C 180,E1 -12885.36,E2 -12885.36} C_VEL
LIN {X 0,Y 312.607,Z 743.939,A -85,B 0,C 180,E1 -12888.203,E2 -12888.203} C_VEL
LIN {X 0,Y 312.265,Z 747.451,A -85,B 0,C 180,E1 -12891.285,E2 -12891.285} C_VEL
LIN {X 0,Y 312.168,Z 749.028,A -85,B 0,C 180,E1 -12894.201,E2 -12894.201} C_VEL
LIN {X 0,Y 312.206,Z 748.828,A -85,B 0,C 180,E1 -12897.253,E2 -12897.253} C_VEL
LIN {X 0,Y 312.438,Z 746.912,A -85,B 0,C 180,E1 -12900.224,E2 -12900.224} C_VEL
LIN {X 0,Y 312.956,Z 743.159,A -85,B 0,C 180,E1 -12903.167,E2 -12903.167} C_VEL
LIN {X 0,Y 313.904,Z 737.534,A -85,B 0,C 180,E1 -12906.102,E2 -12906.102} C_VEL
LIN {X 0,Y 315.295,Z 730.063,A -85,B 0,C 180,E1 -12908.892,E2 -12908.892} C_VEL
LIN {X 0,Y 316.967,Z 721.566,A -85,B 0,C 180,E1 -12911.342,E2 -12911.342} C_VEL
LIN {X 0,Y 319.018,Z 711.003,A -85,B 0,C 180,E1 -12913.713,E2 -12913.713} C_VEL
LIN {X 0,Y 321.176,Z 699.388,A -85,B 0,C 180,E1 -12915.785,E2 -12915.785} C_VEL
LIN {X 0,Y 323.403,Z 686.141,A -85,B 0,C 180,E1 -12917.635,E2 -12917.635} C_VEL
LIN {X 0,Y 325.505,Z 671.84,A -85,B 0,C 180,E1 -12919.199,E2 -12919.199} C_VEL
LIN {X 0,Y 327.266,Z 657.034,A -85,B 0,C 180,E1 -12920.418,E2 -12920.418} C_VEL
LIN {X 0,Y 328.688,Z 641.061,A -85,B 0,C 180,E1 -12921.382,E2 -12921.382} C_VEL
LIN {X 0,Y 329.594,Z 624.254,A -85,B 0,C 180,E1 -12922.032,E2 -12922.032} C_VEL
LIN {X 0,Y 333.422,Z 501.812,A -85,B 0,C 180,E1 -12924.793,E2 -12924.793} C_VEL
LIN {X 0,Y 331.425,Z 482.705,A -85,B 0,C 180,E1 -12925.551,E2 -12925.551} C_VEL
LIN {X 0,Y 335.442,Z 437.528,A -85,B 0,C 180,E1 -12930.152,E2 -12930.152} C_VEL
LIN {X 0,Y 338.999,Z 399.053,A -85,B 0,C 180,E1 -12934.033,E2 -12934.033} C_VEL
LIN {X 0,Y 342.306,Z 362.127,A -85,B 0,C 180,E1 -12937.751,E2 -12937.751} C_VEL
LIN {X 0,Y 337.591,Z 346.974,A -85,B 0,C 180,E1 -12940.266,E2 -12940.266} C_VEL
LIN {X 0,Y 332.324,Z 333.278,A -85,B 0,C 180,E1 -12942.851,E2 -12942.851} C_VEL
LIN {X 0,Y 326.437,Z 320.297,A -85,B 0,C 180,E1 -12945.634,E2 -12945.634} C_VEL
LIN {X 0,Y 321.45,Z 310.966,A -85,B 0,C 180,E1 -12947.971,E2 -12947.971} C_VEL
LIN {X 0,Y 319.417,Z 307.063,A -85,B 0,C 180,E1 -12948.991,E2 -12948.991} C_VEL
LIN {X 0,Y 317.338,Z 303.417,A -85,B 0,C 180,E1 -12950.02,E2 -12950.02} C_VEL
LIN {X 0,Y 316.226,Z 301.786,A -85,B 0,C 180,E1 -12950.536,E2 -12950.536} C_VEL
LIN {X 0,Y 314.376,Z 298.507,A -85,B 0,C 180,E1 -12951.522,E2 -12951.522} C_VEL
LIN {X 0,Y 314.155,Z 297.393,A -85,B 0,C 180,E1 -12952.041,E2 -12952.041} C_VEL
LIN {X 0,Y 314.165,Z 297.347,A -85,B 0,C 180,E1 -12956.533,E2 -12956.533} C_VEL
LIN {X 0,Y 314.171,Z 297.344,A -85,B 0,C 180,E1 -12960.911,E2 -12960.911} C_VEL
LIN {X 0,Y 314.151,Z 297.354,A -85,B 0,C 180,E1 -12965.478,E2 -12965.478} C_VEL
LIN {X 0,Y 314.146,Z 297.345,A -85,B 0,C 180,E1 -12969.896,E2 -12969.896} C_VEL
LIN {X 0,Y 314.161,Z 297.354,A -85,B 0,C 180,E1 -12974.373,E2 -12974.373} C_VEL
LIN {X 0,Y 314.17,Z 297.343,A -85,B 0,C 180,E1 -12978.749,E2 -12978.749} C_VEL
LIN {X 0,Y 314.172,Z 297.351,A -85,B 0,C 180,E1 -12983.242,E2 -12983.242} C_VEL
LIN {X 0,Y 314.155,Z 297.349,A -85,B 0,C 180,E1 -12987.78,E2 -12987.78} C_VEL
LIN {X 0,Y 314.207,Z 297.632,A -85,B 0,C 180,E1 -12991.457,E2 -12991.457} C_VEL
LIN {X 0,Y 315.623,Z 301.081,A -85,B 0,C 180,E1 -12992.369,E2 -12992.369} C_VEL
LIN {X 0,Y 322.969,Z 317.218,A -85,B 0,C 180,E1 -12996.249,E2 -12996.249} C_VEL
LIN {X 0,Y 325.12,Z 321.958,A -85,B 0,C 180,E1 -12997.234,E2 -12997.234} C_VEL
LIN {X 0,Y 339.923,Z 346.539,A -85,B 0,C 180,E1 -13000.407,E2 -13000.407} C_VEL
LIN {X 0,Y 354.859,Z 373.04,A -85,B 0,C 180,E1 -13003.321,E2 -13003.321} C_VEL
LIN {X 0,Y 356.871,Z 377.15,A -85,B 0,C 180,E1 -13003.709,E2 -13003.709} C_VEL
LIN {X 0,Y 344.034,Z 576.734,A -85,B 0,C 180,E1 -13008.907,E2 -13008.907} C_VEL
LIN {X 0,Y 341.881,Z 598.232,A -85,B 0,C 180,E1 -13009.757,E2 -13009.757} C_VEL
LIN {X 0,Y 339.198,Z 619.151,A -85,B 0,C 180,E1 -13010.893,E2 -13010.893} C_VEL
LIN {X 0,Y 336.079,Z 639.65,A -85,B 0,C 180,E1 -13012.345,E2 -13012.345} C_VEL
LIN {X 0,Y 332.807,Z 658.657,A -85,B 0,C 180,E1 -13014.034,E2 -13014.034} C_VEL
LIN {X 0,Y 329.239,Z 677.46,A -85,B 0,C 180,E1 -13016.092,E2 -13016.092} C_VEL
LIN {X 0,Y 325.708,Z 695.046,A -85,B 0,C 180,E1 -13018.442,E2 -13018.442} C_VEL
LIN {X 0,Y 322.353,Z 711.252,A -85,B 0,C 180,E1 -13021.064,E2 -13021.064} C_VEL
LIN {X 0,Y 319.275,Z 726.233,A -85,B 0,C 180,E1 -13023.999,E2 -13023.999} C_VEL
LIN {X 0,Y 316.82,Z 738.788,A -85,B 0,C 180,E1 -13026.965,E2 -13026.965} C_VEL
LIN {X 0,Y 314.859,Z 749.859,A -85,B 0,C 180,E1 -13030.139,E2 -13030.139} C_VEL
LIN {X 0,Y 313.501,Z 758.929,A -85,B 0,C 180,E1 -13033.321,E2 -13033.321} C_VEL
LIN {X 0,Y 312.614,Z 766.626,A -85,B 0,C 180,E1 -13036.688,E2 -13036.688} C_VEL
LIN {X 0,Y 312.189,Z 772.809,A -85,B 0,C 180,E1 -13040.229,E2 -13040.229} C_VEL
LIN {X 0,Y 312.1,Z 776.968,A -85,B 0,C 180,E1 -13043.564,E2 -13043.564} C_VEL
LIN {X 0,Y 312.119,Z 779.473,A -85,B 0,C 180,E1 -13046.88,E2 -13046.88} C_VEL
LIN {X 0,Y 312.146,Z 780.41,A -85,B 0,C 180,E1 -13050.186,E2 -13050.186} C_VEL
LIN {X 0,Y 312.083,Z 779.858,A -85,B 0,C 180,E1 -13053.492,E2 -13053.492} C_VEL
LIN {X 0,Y 312.051,Z 777.77,A -85,B 0,C 180,E1 -13056.811,E2 -13056.811} C_VEL
LIN {X 0,Y 312.18,Z 774.12,A -85,B 0,C 180,E1 -13060.148,E2 -13060.148} C_VEL
LIN {X 0,Y 312.695,Z 768.613,A -85,B 0,C 180,E1 -13063.689,E2 -13063.689} C_VEL
LIN {X 0,Y 313.732,Z 761.756,A -85,B 0,C 180,E1 -13067.052,E2 -13067.052} C_VEL
LIN {X 0,Y 315.522,Z 752.593,A -85,B 0,C 180,E1 -13070.596,E2 -13070.596} C_VEL
LIN {X 0,Y 318.153,Z 741.278,A -85,B 0,C 180,E1 -13074.116,E2 -13074.116} C_VEL
LIN {X 0,Y 321.514,Z 728.328,A -85,B 0,C 180,E1 -13077.405,E2 -13077.405} C_VEL
LIN {X 0,Y 325.509,Z 713.816,A -85,B 0,C 180,E1 -13080.454,E2 -13080.454} C_VEL
LIN {X 0,Y 330.18,Z 697.464,A -85,B 0,C 180,E1 -13083.303,E2 -13083.303} C_VEL
LIN {X 0,Y 335.464,Z 679.029,A -85,B 0,C 180,E1 -13085.958,E2 -13085.958} C_VEL
LIN {X 0,Y 340.919,Z 659.877,A -85,B 0,C 180,E1 -13088.232,E2 -13088.232} C_VEL
LIN {X 0,Y 346.959,Z 638.42,A -85,B 0,C 180,E1 -13090.314,E2 -13090.314} C_VEL
LIN {X 0,Y 353.072,Z 616.191,A -85,B 0,C 180,E1 -13092.049,E2 -13092.049} C_VEL
LIN {X 0,Y 358.873,Z 594.337,A -85,B 0,C 180,E1 -13093.377,E2 -13093.377} C_VEL
LIN {X 0,Y 364.617,Z 570.641,A -85,B 0,C 180,E1 -13094.466,E2 -13094.466} C_VEL
LIN {X 0,Y 377.031,Z 516.92,A -85,B 0,C 180,E1 -13096.468,E2 -13096.468} C_VEL
LIN {X 0,Y 381.467,Z 500.047,A -85,B 0,C 180,E1 -13097.105,E2 -13097.105} C_VEL
LIN {X 0,Y 366.445,Z 559.755,A -85,B 0,C 180,E1 -13099.415,E2 -13099.415} C_VEL
LIN {X 0,Y 360.935,Z 581.963,A -85,B 0,C 180,E1 -13100.421,E2 -13100.421} C_VEL
LIN {X 0,Y 355.075,Z 603.113,A -85,B 0,C 180,E1 -13101.721,E2 -13101.721} C_VEL
LIN {X 0,Y 348.859,Z 624.354,A -85,B 0,C 180,E1 -13103.406,E2 -13103.406} C_VEL
LIN {X 0,Y 342.955,Z 643.935,A -85,B 0,C 180,E1 -13105.354,E2 -13105.354} C_VEL
LIN {X 0,Y 337.175,Z 662.515,A -85,B 0,C 180,E1 -13107.639,E2 -13107.639} C_VEL
LIN {X 0,Y 331.809,Z 679.598,A -85,B 0,C 180,E1 -13110.212,E2 -13110.212} C_VEL
LIN {X 0,Y 327.161,Z 694.304,A -85,B 0,C 180,E1 -13112.912,E2 -13112.912} C_VEL
LIN {X 0,Y 323.006,Z 707.545,A -85,B 0,C 180,E1 -13115.883,E2 -13115.883} C_VEL
LIN {X 0,Y 319.633,Z 718.492,A -85,B 0,C 180,E1 -13118.917,E2 -13118.917} C_VEL
LIN {X 0,Y 316.864,Z 727.897,A -85,B 0,C 180,E1 -13122.177,E2 -13122.177} C_VEL
LIN {X 0,Y 314.86,Z 735.32,A -85,B 0,C 180,E1 -13125.472,E2 -13125.472} C_VEL
LIN {X 0,Y 313.523,Z 740.919,A -85,B 0,C 180,E1 -13128.783,E2 -13128.783} C_VEL
LIN {X 0,Y 312.721,Z 744.807,A -85,B 0,C 180,E1 -13132.098,E2 -13132.098} C_VEL
LIN {X 0,Y 312.307,Z 747.109,A -85,B 0,C 180,E1 -13135.594,E2 -13135.594} C_VEL
LIN {X 0,Y 312.167,Z 747.631,A -85,B 0,C 180,E1 -13138.899,E2 -13138.899} C_VEL
LIN {X 0,Y 312.123,Z 746.506,A -85,B 0,C 180,E1 -13142.204,E2 -13142.204} C_VEL
LIN {X 0,Y 312.205,Z 743.731,A -85,B 0,C 180,E1 -13145.514,E2 -13145.514} C_VEL
LIN {X 0,Y 312.502,Z 739.236,A -85,B 0,C 180,E1 -13148.835,E2 -13148.835} C_VEL
LIN {X 0,Y 313.109,Z 733.292,A -85,B 0,C 180,E1 -13151.98,E2 -13151.98} C_VEL
LIN {X 0,Y 314.157,Z 725.57,A -85,B 0,C 180,E1 -13155.129,E2 -13155.129} C_VEL
LIN {X 0,Y 315.737,Z 715.857,A -85,B 0,C 180,E1 -13158.272,E2 -13158.272} C_VEL
LIN {X 0,Y 317.776,Z 704.613,A -85,B 0,C 180,E1 -13161.214,E2 -13161.214} C_VEL
LIN {X 0,Y 320.217,Z 691.886,A -85,B 0,C 180,E1 -13163.949,E2 -13163.949} C_VEL
LIN {X 0,Y 322.985,Z 677.669,A -85,B 0,C 180,E1 -13166.474,E2 -13166.474} C_VEL
LIN {X 0,Y 325.992,Z 661.889,A -85,B 0,C 180,E1 -13168.787,E2 -13168.787} C_VEL
LIN {X 0,Y 329.153,Z 644.286,A -85,B 0,C 180,E1 -13170.889,E2 -13170.889} C_VEL
LIN {X 0,Y 332.082,Z 626.513,A -85,B 0,C 180,E1 -13172.613,E2 -13172.613} C_VEL
LIN {X 0,Y 334.806,Z 607.979,A -85,B 0,C 180,E1 -13174.053,E2 -13174.053} C_VEL
LIN {X 0,Y 337.196,Z 588.684,A -85,B 0,C 180,E1 -13175.222,E2 -13175.222} C_VEL
LIN {X 0,Y 339.331,Z 567.495,A -85,B 0,C 180,E1 -13176.159,E2 -13176.159} C_VEL
LIN {X 0,Y 341.441,Z 536.028,A -85,B 0,C 180,E1 -13177.09,E2 -13177.09} C_VEL
LIN {X 0,Y 351.309,Z 385.374,A -85,B 0,C 180,E1 -13181.187,E2 -13181.187} C_VEL
LIN {X 0,Y 349.678,Z 373.169,A -85,B 0,C 180,E1 -13181.82,E2 -13181.82} C_VEL
LIN {X 0,Y 335.154,Z 345.914,A -85,B 0,C 180,E1 -13184.731,E2 -13184.731} C_VEL
LIN {X 0,Y 330.764,Z 337.858,A -85,B 0,C 180,E1 -13185.709,E2 -13185.709} C_VEL
LIN {X 0,Y 323.739,Z 320.175,A -85,B 0,C 180,E1 -13189.564,E2 -13189.564} C_VEL
LIN {X 0,Y 317.35,Z 304.98,A -85,B 0,C 180,E1 -13193.227,E2 -13193.227} C_VEL
LIN {X 0,Y 314.204,Z 297.608,A -85,B 0,C 180,E1 -13195.187,E2 -13195.187} C_VEL
LIN {X 0,Y 314.174,Z 297.326,A -85,B 0,C 180,E1 -13199.599,E2 -13199.599} C_VEL
LIN {X 0,Y 314.192,Z 297.569,A -85,B 0,C 180,E1 -13201.174,E2 -13201.174} C_VEL
LIN {X 0,Y 315.268,Z 300.467,A -85,B 0,C 180,E1 -13201.846,E2 -13201.846} C_VEL
LIN {X 0,Y 316.442,Z 302.54,A -85,B 0,C 180,E1 -13202.322,E2 -13202.322} C_VEL
LIN {X 0,Y 323.43,Z 317.197,A -85,B 0,C 180,E1 -13205.353,E2 -13205.353} C_VEL
LIN {X 0,Y 330.61,Z 334.343,A -85,B 0,C 180,E1 -13208.533,E2 -13208.533} C_VEL
LIN {X 0,Y 336.995,Z 352.041,A -85,B 0,C 180,E1 -13211.488,E2 -13211.488} C_VEL
LIN {X 0,Y 339.833,Z 361.857,A -85,B 0,C 180,E1 -13212.986,E2 -13212.986} C_VEL
LIN {X 0,Y 336.205,Z 402.075,A -85,B 0,C 180,E1 -13217.11,E2 -13217.11} C_VEL
LIN {X 0,Y 332.629,Z 441.744,A -85,B 0,C 180,E1 -13221.18,E2 -13221.18} C_VEL
LIN {X 0,Y 329.266,Z 482.332,A -85,B 0,C 180,E1 -13225.317,E2 -13225.317} C_VEL
LIN {X 0,Y 331.319,Z 504.222,A -85,B 0,C 180,E1 -13226.048,E2 -13226.048} C_VEL
LIN {X 0,Y 327.654,Z 626.241,A -85,B 0,C 180,E1 -13228.774,E2 -13228.774} C_VEL
LIN {X 0,Y 327.484,Z 629.952,A -85,B 0,C 180,E1 -13228.905,E2 -13228.905} C_VEL
LIN {X 0,Y 325.817,Z 638.541,A -85,B 0,C 180,E1 -13229.168,E2 -13229.168} C_VEL
LIN {X 0,Y 319.849,Z 653.981,A -85,B 0,C 180,E1 -13229.671,E2 -13229.671} C_VEL
LIN {X 0,Y 317.824,Z 661.131,A -85,B 0,C 180,E1 -13230.099,E2 -13230.099} C_VEL
LIN {X 0,Y 317.518,Z 663.107,A -85,B 0,C 180,E1 -13230.255,E2 -13230.255} C_VEL
LIN {X 0,Y 315.7,Z 677.597,A -85,B 0,C 180,E1 -13231.631,E2 -13231.631} C_VEL
LIN {X 0,Y 313.688,Z 691.008,A -85,B 0,C 180,E1 -13233.287,E2 -13233.287} C_VEL
LIN {X 0,Y 311.602,Z 703.615,A -85,B 0,C 180,E1 -13235.249,E2 -13235.249} C_VEL
LIN {X 0,Y 309.591,Z 714.862,A -85,B 0,C 180,E1 -13237.473,E2 -13237.473} C_VEL
LIN {X 0,Y 307.812,Z 724.685,A -85,B 0,C 180,E1 -13239.911,E2 -13239.911} C_VEL
LIN {X 0,Y 306.314,Z 733.152,A -85,B 0,C 180,E1 -13242.63,E2 -13242.63} C_VEL
LIN {X 0,Y 305.271,Z 739.69,A -85,B 0,C 180,E1 -13245.382,E2 -13245.382} C_VEL
LIN {X 0,Y 304.625,Z 744.461,A -85,B 0,C 180,E1 -13248.166,E2 -13248.166} C_VEL
LIN {X 0,Y 304.281,Z 747.806,A -85,B 0,C 180,E1 -13251.187,E2 -13251.187} C_VEL
LIN {X 0,Y 304.177,Z 749.381,A -85,B 0,C 180,E1 -13254.052,E2 -13254.052} C_VEL
LIN {X 0,Y 304.209,Z 749.326,A -85,B 0,C 180,E1 -13257.036,E2 -13257.036} C_VEL
LIN {X 0,Y 304.444,Z 747.509,A -85,B 0,C 180,E1 -13260.162,E2 -13260.162} C_VEL
LIN {X 0,Y 304.981,Z 743.907,A -85,B 0,C 180,E1 -13263.193,E2 -13263.193} C_VEL
LIN {X 0,Y 305.985,Z 738.311,A -85,B 0,C 180,E1 -13266.257,E2 -13266.257} C_VEL
LIN {X 0,Y 307.351,Z 731.431,A -85,B 0,C 180,E1 -13268.966,E2 -13268.966} C_VEL
LIN {X 0,Y 309.223,Z 722.437,A -85,B 0,C 180,E1 -13271.674,E2 -13271.674} C_VEL
LIN {X 0,Y 311.258,Z 712.593,A -85,B 0,C 180,E1 -13273.981,E2 -13273.981} C_VEL
LIN {X 0,Y 313.635,Z 700.469,A -85,B 0,C 180,E1 -13276.227,E2 -13276.227} C_VEL
LIN {X 0,Y 315.884,Z 687.906,A -85,B 0,C 180,E1 -13278.056,E2 -13278.056} C_VEL
LIN {X 0,Y 318.138,Z 673.471,A -85,B 0,C 180,E1 -13279.702,E2 -13279.702} C_VEL
LIN {X 0,Y 320.016,Z 658.803,A -85,B 0,C 180,E1 -13280.969,E2 -13280.969} C_VEL
LIN {X 0,Y 321.584,Z 642.411,A -85,B 0,C 180,E1 -13282.002,E2 -13282.002} C_VEL
LIN {X 0,Y 322.547,Z 626.195,A -85,B 0,C 180,E1 -13282.668,E2 -13282.668} C_VEL
LIN {X 0,Y 326.646,Z 502.725,A -85,B 0,C 180,E1 -13285.521,E2 -13285.521} C_VEL
LIN {X 0,Y 324.633,Z 483.021,A -85,B 0,C 180,E1 -13286.33,E2 -13286.33} C_VEL
LIN {X 0,Y 328.77,Z 438.859,A -85,B 0,C 180,E1 -13290.882,E2 -13290.882} C_VEL
LIN {X 0,Y 332.769,Z 398.4,A -85,B 0,C 180,E1 -13295.029,E2 -13295.029} C_VEL
LIN {X 0,Y 335.797,Z 365.098,A -85,B 0,C 180,E1 -13298.424,E2 -13298.424} C_VEL
LIN {X 0,Y 331.194,Z 350.272,A -85,B 0,C 180,E1 -13300.97,E2 -13300.97} C_VEL
LIN {X 0,Y 326.01,Z 336.794,A -85,B 0,C 180,E1 -13303.61,E2 -13303.61} C_VEL
LIN {X 0,Y 320.64,Z 324.896,A -85,B 0,C 180,E1 -13306.29,E2 -13306.29} C_VEL
LIN {X 0,Y 316.472,Z 316.888,A -85,B 0,C 180,E1 -13308.339,E2 -13308.339} C_VEL
LIN {X 0,Y 314.082,Z 312.525,A -85,B 0,C 180,E1 -13309.545,E2 -13309.545} C_VEL
LIN {X 0,Y 311.75,Z 308.29,A -85,B 0,C 180,E1 -13310.771,E2 -13310.771} C_VEL
LIN {X 0,Y 309.749,Z 304.971,A -85,B 0,C 180,E1 -13311.834,E2 -13311.834} C_VEL
LIN {X 0,Y 308.797,Z 303.284,A -85,B 0,C 180,E1 -13312.371,E2 -13312.371} C_VEL
LIN {X 0,Y 306.75,Z 300.399,A -85,B 0,C 180,E1 -13313.449,E2 -13313.449} C_VEL
LIN {X 0,Y 306.26,Z 298.675,A -85,B 0,C 180,E1 -13314.003,E2 -13314.003} C_VEL
LIN {X 0,Y 306.207,Z 298.337,A -85,B 0,C 180,E1 -13315.88,E2 -13315.88} C_VEL
LIN {X 0,Y 306.224,Z 298.337,A -85,B 0,C 180,E1 -13320.373,E2 -13320.373} C_VEL
LIN {X 0,Y 306.231,Z 298.337,A -85,B 0,C 180,E1 -13324.869,E2 -13324.869} C_VEL
LIN {X 0,Y 306.222,Z 298.333,A -85,B 0,C 180,E1 -13329.206,E2 -13329.206} C_VEL
LIN {X 0,Y 306.208,Z 298.34,A -85,B 0,C 180,E1 -13333.789,E2 -13333.789} C_VEL
LIN {X 0,Y 306.215,Z 298.335,A -85,B 0,C 180,E1 -13338.267,E2 -13338.267} C_VEL
LIN {X 0,Y 306.244,Z 298.334,A -85,B 0,C 180,E1 -13342.862,E2 -13342.862} C_VEL
LIN {X 0,Y 306.226,Z 298.335,A -85,B 0,C 180,E1 -13347.411,E2 -13347.411} C_VEL
LIN {X 0,Y 306.246,Z 298.564,A -85,B 0,C 180,E1 -13350.04,E2 -13350.04} C_VEL
LIN {X 0,Y 307.852,Z 302.276,A -85,B 0,C 180,E1 -13351.091,E2 -13351.091} C_VEL
LIN {X 0,Y 315.057,Z 318.13,A -85,B 0,C 180,E1 -13355.058,E2 -13355.058} C_VEL
LIN {X 0,Y 316.939,Z 322.177,A -85,B 0,C 180,E1 -13355.928,E2 -13355.928} C_VEL
LIN {X 0,Y 332.048,Z 347.169,A -85,B 0,C 180,E1 -13359.307,E2 -13359.307} C_VEL
LIN {X 0,Y 347.478,Z 374.403,A -85,B 0,C 180,E1 -13362.436,E2 -13362.436} C_VEL
LIN {X 0,Y 350.314,Z 380.038,A -85,B 0,C 180,E1 -13362.993,E2 -13362.993} C_VEL
LIN {X 0,Y 337.058,Z 576.643,A -85,B 0,C 180,E1 -13368.247,E2 -13368.247} C_VEL
LIN {X 0,Y 334.887,Z 597.608,A -85,B 0,C 180,E1 -13369.089,E2 -13369.089} C_VEL
LIN {X 0,Y 332.084,Z 618.839,A -85,B 0,C 180,E1 -13370.262,E2 -13370.262} C_VEL
LIN {X 0,Y 328.838,Z 639.488,A -85,B 0,C 180,E1 -13371.753,E2 -13371.753} C_VEL
LIN {X 0,Y 325.379,Z 658.903,A -85,B 0,C 180,E1 -13373.518,E2 -13373.518} C_VEL
LIN {X 0,Y 321.792,Z 677.22,A -85,B 0,C 180,E1 -13375.566,E2 -13375.566} C_VEL
LIN {X 0,Y 318.199,Z 694.568,A -85,B 0,C 180,E1 -13377.927,E2 -13377.927} C_VEL
LIN {X 0,Y 314.704,Z 710.893,A -85,B 0,C 180,E1 -13380.62,E2 -13380.62} C_VEL
LIN {X 0,Y 311.588,Z 725.552,A -85,B 0,C 180,E1 -13383.544,E2 -13383.544} C_VEL
LIN {X 0,Y 308.91,Z 738.785,A -85,B 0,C 180,E1 -13386.744,E2 -13386.744} C_VEL
LIN {X 0,Y 306.797,Z 750.422,A -85,B 0,C 180,E1 -13390.19,E2 -13390.19} C_VEL
LIN {X 0,Y 305.379,Z 759.821,A -85,B 0,C 180,E1 -13393.648,E2 -13393.648} C_VEL
LIN {X 0,Y 304.527,Z 767.412,A -85,B 0,C 180,E1 -13397.197,E2 -13397.197} C_VEL
LIN {X 0,Y 304.178,Z 772.851,A -85,B 0,C 180,E1 -13400.542,E2 -13400.542} C_VEL
LIN {X 0,Y 304.115,Z 776.821,A -85,B 0,C 180,E1 -13403.963,E2 -13403.963} C_VEL
LIN {X 0,Y 304.142,Z 779.211,A -85,B 0,C 180,E1 -13407.364,E2 -13407.364} C_VEL
LIN {X 0,Y 304.153,Z 779.937,A -85,B 0,C 180,E1 -13410.567,E2 -13410.567} C_VEL
LIN {X 0,Y 304.087,Z 779.271,A -85,B 0,C 180,E1 -13413.961,E2 -13413.961} C_VEL
LIN {X 0,Y 304.051,Z 777.109,A -85,B 0,C 180,E1 -13417.37,E2 -13417.37} C_VEL
LIN {X 0,Y 304.261,Z 773.101,A -85,B 0,C 180,E1 -13420.99,E2 -13420.99} C_VEL
LIN {X 0,Y 304.947,Z 767.241,A -85,B 0,C 180,E1 -13424.707,E2 -13424.707} C_VEL
LIN {X 0,Y 306.34,Z 759.409,A -85,B 0,C 180,E1 -13428.459,E2 -13428.459} C_VEL
LIN {X 0,Y 308.517,Z 749.839,A -85,B 0,C 180,E1 -13432.084,E2 -13432.084} C_VEL
LIN {X 0,Y 311.541,Z 738.368,A -85,B 0,C 180,E1 -13435.6,E2 -13435.6} C_VEL
LIN {X 0,Y 315.243,Z 725.575,A -85,B 0,C 180,E1 -13438.824,E2 -13438.824} C_VEL
LIN {X 0,Y 319.739,Z 710.854,A -85,B 0,C 180,E1 -13441.905,E2 -13441.905} C_VEL
LIN {X 0,Y 324.84,Z 694.576,A -85,B 0,C 180,E1 -13444.733,E2 -13444.733} C_VEL
LIN {X 0,Y 330.567,Z 676.536,A -85,B 0,C 180,E1 -13447.335,E2 -13447.335} C_VEL
LIN {X 0,Y 337.026,Z 656.216,A -85,B 0,C 180,E1 -13449.743,E2 -13449.743} C_VEL
LIN {X 0,Y 343.944,Z 634.344,A -85,B 0,C 180,E1 -13451.85,E2 -13451.85} C_VEL
LIN {X 0,Y 350.732,Z 612.655,A -85,B 0,C 180,E1 -13453.51,E2 -13453.51} C_VEL
LIN {X 0,Y 357.072,Z 591.467,A -85,B 0,C 180,E1 -13454.77,E2 -13454.77} C_VEL
LIN {X 0,Y 363.788,Z 566.83,A -85,B 0,C 180,E1 -13455.866,E2 -13455.866} C_VEL
LIN {X 0,Y 372.301,Z 533.607,A -85,B 0,C 180,E1 -13457.126,E2 -13457.126} C_VEL
LIN {X 0,Y 360.852,Z 576.04,A -85,B 0,C 180,E1 -13458.848,E2 -13458.848} C_VEL
LIN {X 0,Y 354.598,Z 596.497,A -85,B 0,C 180,E1 -13459.993,E2 -13459.993} C_VEL
LIN {X 0,Y 347.835,Z 617.125,A -85,B 0,C 180,E1 -13461.514,E2 -13461.514} C_VEL
LIN {X 0,Y 341.059,Z 637.015,A -85,B 0,C 180,E1 -13463.375,E2 -13463.375} C_VEL
LIN {X 0,Y 334.362,Z 656.332,A -85,B 0,C 180,E1 -13465.625,E2 -13465.625} C_VEL
LIN {X 0,Y 328.316,Z 673.71,A -85,B 0,C 180,E1 -13468.105,E2 -13468.105} C_VEL
LIN {X 0,Y 322.738,Z 689.716,A -85,B 0,C 180,E1 -13470.897,E2 -13470.897} C_VEL
LIN {X 0,Y 317.877,Z 703.571,A -85,B 0,C 180,E1 -13473.874,E2 -13473.874} C_VEL
LIN {X 0,Y 313.881,Z 715.175,A -85,B 0,C 180,E1 -13476.933,E2 -13476.933} C_VEL
LIN {X 0,Y 310.524,Z 725.268,A -85,B 0,C 180,E1 -13480.24,E2 -13480.24} C_VEL
LIN {X 0,Y 308.003,Z 733.339,A -85,B 0,C 180,E1 -13483.596,E2 -13483.596} C_VEL
LIN {X 0,Y 306.161,Z 739.845,A -85,B 0,C 180,E1 -13487.17,E2 -13487.17} C_VEL
LIN {X 0,Y 305.03,Z 744.424,A -85,B 0,C 180,E1 -13490.758,E2 -13490.758} C_VEL
LIN {X 0,Y 304.445,Z 747.163,A -85,B 0,C 180,E1 -13494.346,E2 -13494.346} C_VEL
LIN {X 0,Y 304.206,Z 748.1,A -85,B 0,C 180,E1 -13497.74,E2 -13497.74} C_VEL
LIN {X 0,Y 304.14,Z 747.413,A -85,B 0,C 180,E1 -13501.131,E2 -13501.131} C_VEL
LIN {X 0,Y 304.167,Z 745.086,A -85,B 0,C 180,E1 -13504.526,E2 -13504.526} C_VEL
LIN {X 0,Y 304.381,Z 741.334,A -85,B 0,C 180,E1 -13507.741,E2 -13507.741} C_VEL
LIN {X 0,Y 304.928,Z 735.584,A -85,B 0,C 180,E1 -13511.156,E2 -13511.156} C_VEL
LIN {X 0,Y 305.866,Z 728.363,A -85,B 0,C 180,E1 -13514.386,E2 -13514.386} C_VEL
LIN {X 0,Y 307.335,Z 719.193,A -85,B 0,C 180,E1 -13517.612,E2 -13517.612} C_VEL
LIN {X 0,Y 309.278,Z 708.546,A -85,B 0,C 180,E1 -13520.634,E2 -13520.634} C_VEL
LIN {X 0,Y 311.636,Z 696.489,A -85,B 0,C 180,E1 -13523.444,E2 -13523.444} C_VEL
LIN {X 0,Y 314.332,Z 683.05,A -85,B 0,C 180,E1 -13526.039,E2 -13526.039} C_VEL
LIN {X 0,Y 317.368,Z 667.769,A -85,B 0,C 180,E1 -13528.477,E2 -13528.477} C_VEL
LIN {X 0,Y 320.536,Z 651.099,A -85,B 0,C 180,E1 -13530.665,E2 -13530.665} C_VEL
LIN {X 0,Y 323.76,Z 632.878,A -85,B 0,C 180,E1 -13532.61,E2 -13532.61} C_VEL
LIN {X 0,Y 326.7,Z 614.266,A -85,B 0,C 180,E1 -13534.205,E2 -13534.205} C_VEL
LIN {X 0,Y 329.424,Z 594.374,A -85,B 0,C 180,E1 -13535.538,E2 -13535.538} C_VEL
LIN {X 0,Y 331.752,Z 573.477,A -85,B 0,C 180,E1 -13536.584,E2 -13536.584} C_VEL
LIN {X 0,Y 333.538,Z 551.332,A -85,B 0,C 180,E1 -13537.336,E2 -13537.336} C_VEL
LIN {X 0,Y 344.781,Z 386.537,A -85,B 0,C 180,E1 -13541.938,E2 -13541.938} C_VEL
LIN {X 0,Y 343.509,Z 376.898,A -85,B 0,C 180,E1 -13542.448,E2 -13542.448} C_VEL
LIN {X 0,Y 329.817,Z 350.976,A -85,B 0,C 180,E1 -13545.274,E2 -13545.274} C_VEL
LIN {X 0,Y 322.394,Z 337.465,A -85,B 0,C 180,E1 -13546.975,E2 -13546.975} C_VEL
LIN {X 0,Y 315.826,Z 320.992,A -85,B 0,C 180,E1 -13550.714,E2 -13550.714} C_VEL
LIN {X 0,Y 309.267,Z 305.717,A -85,B 0,C 180,E1 -13554.561,E2 -13554.561} C_VEL
LIN {X 0,Y 306.256,Z 298.499,A -85,B 0,C 180,E1 -13556.573,E2 -13556.573} C_VEL
LIN {X 0,Y 306.266,Z 298.491,A -85,B 0,C 180,E1 -13559.761,E2 -13559.761} C_VEL
LIN {X 0,Y 306.625,Z 299.95,A -85,B 0,C 180,E1 -13560.158,E2 -13560.158} C_VEL
LIN {X 0,Y 308.818,Z 304.202,A -85,B 0,C 180,E1 -13561.155,E2 -13561.155} C_VEL
LIN {X 0,Y 315.036,Z 316.957,A -85,B 0,C 180,E1 -13563.922,E2 -13563.922} C_VEL
LIN {X 0,Y 321.803,Z 332.294,A -85,B 0,C 180,E1 -13566.951,E2 -13566.951} C_VEL
LIN {X 0,Y 328.534,Z 350.253,A -85,B 0,C 180,E1 -13570.123,E2 -13570.123} C_VEL
LIN {X 0,Y 332.994,Z 364.788,A -85,B 0,C 180,E1 -13572.435,E2 -13572.435} C_VEL
LIN {X 0,Y 328.99,Z 407.138,A -85,B 0,C 180,E1 -13576.823,E2 -13576.823} C_VEL
LIN {X 0,Y 324.968,Z 450.502,A -85,B 0,C 180,E1 -13581.327,E2 -13581.327} C_VEL
LIN {X 0,Y 322.15,Z 482.695,A -85,B 0,C 180,E1 -13584.65,E2 -13584.65} C_VEL
LIN {X 0,Y 324.203,Z 504.951,A -85,B 0,C 180,E1 -13585.416,E2 -13585.416} C_VEL
LIN {X 0,Y 320.395,Z 626.529,A -85,B 0,C 180,E1 -13588.182,E2 -13588.182} C_VEL
LIN {X 0,Y 319.442,Z 642.663,A -85,B 0,C 180,E1 -13588.874,E2 -13588.874} C_VEL
LIN {X 0,Y 318.04,Z 658.371,A -85,B 0,C 180,E1 -13589.878,E2 -13589.878} C_VEL
LIN {X 0,Y 317.518,Z 663.107,A -85,B 0,C 180,E1 -13590.255,E2 -13590.255} C_VEL
LIN {X 0,Y 315.774,Z 670.088,A -85,B 0,C 180,E1 -13590.797,E2 -13590.797} C_VEL
LIN {X 0,Y 309.07,Z 684.144,A -85,B 0,C 180,E1 -13591.955,E2 -13591.955} C_VEL
LIN {X 0,Y 306.269,Z 691.31,A -85,B 0,C 180,E1 -13592.778,E2 -13592.778} C_VEL
LIN {X 0,Y 305.895,Z 693.038,A -85,B 0,C 180,E1 -13593.018,E2 -13593.018} C_VEL
LIN {X 0,Y 303.776,Z 705.14,A -85,B 0,C 180,E1 -13595.002,E2 -13595.002} C_VEL
LIN {X 0,Y 301.589,Z 716.836,A -85,B 0,C 180,E1 -13597.427,E2 -13597.427} C_VEL
LIN {X 0,Y 299.746,Z 726.488,A -85,B 0,C 180,E1 -13599.987,E2 -13599.987} C_VEL
LIN {X 0,Y 298.247,Z 734.68,A -85,B 0,C 180,E1 -13602.781,E2 -13602.781} C_VEL
LIN {X 0,Y 297.213,Z 740.914,A -85,B 0,C 180,E1 -13605.61,E2 -13605.61} C_VEL
LIN {X 0,Y 296.555,Z 745.698,A -85,B 0,C 180,E1 -13608.679,E2 -13608.679} C_VEL
LIN {X 0,Y 296.269,Z 748.563,A -85,B 0,C 180,E1 -13611.581,E2 -13611.581} C_VEL
LIN {X 0,Y 296.18,Z 749.881,A -85,B 0,C 180,E1 -13614.753,E2 -13614.753} C_VEL
LIN {X 0,Y 296.259,Z 749.494,A -85,B 0,C 180,E1 -13617.84,E2 -13617.84} C_VEL
LIN {X 0,Y 296.546,Z 747.466,A -85,B 0,C 180,E1 -13620.827,E2 -13620.827} C_VEL
LIN {X 0,Y 297.199,Z 743.571,A -85,B 0,C 180,E1 -13623.947,E2 -13623.947} C_VEL
LIN {X 0,Y 298.269,Z 738.131,A -85,B 0,C 180,E1 -13626.87,E2 -13626.87} C_VEL
LIN {X 0,Y 299.875,Z 730.609,A -85,B 0,C 180,E1 -13629.802,E2 -13629.802} C_VEL
LIN {X 0,Y 301.777,Z 722.054,A -85,B 0,C 180,E1 -13632.365,E2 -13632.365} C_VEL
LIN {X 0,Y 304.089,Z 711.402,A -85,B 0,C 180,E1 -13634.849,E2 -13634.849} C_VEL
LIN {X 0,Y 306.506,Z 699.659,A -85,B 0,C 180,E1 -13637.016,E2 -13637.016} C_VEL
LIN {X 0,Y 308.971,Z 686.351,A -85,B 0,C 180,E1 -13638.935,E2 -13638.935} C_VEL
LIN {X 0,Y 311.195,Z 672.566,A -85,B 0,C 180,E1 -13640.492,E2 -13640.492} C_VEL
LIN {X 0,Y 313.133,Z 657.699,A -85,B 0,C 180,E1 -13641.763,E2 -13641.763} C_VEL
LIN {X 0,Y 314.68,Z 641.854,A -85,B 0,C 180,E1 -13642.753,E2 -13642.753} C_VEL
LIN {X 0,Y 315.684,Z 624.99,A -85,B 0,C 180,E1 -13643.43,E2 -13643.43} C_VEL
LIN {X 0,Y 319.916,Z 503.512,A -85,B 0,C 180,E1 -13646.285,E2 -13646.285} C_VEL
LIN {X 0,Y 317.902,Z 483.756,A -85,B 0,C 180,E1 -13647.11,E2 -13647.11} C_VEL
LIN {X 0,Y 322.289,Z 439.065,A -85,B 0,C 180,E1 -13651.766,E2 -13651.766} C_VEL
LIN {X 0,Y 326.267,Z 400.494,A -85,B 0,C 180,E1 -13655.754,E2 -13655.754} C_VEL
LIN {X 0,Y 329.455,Z 368.511,A -85,B 0,C 180,E1 -13659.061,E2 -13659.061} C_VEL
LIN {X 0,Y 324.873,Z 353.638,A -85,B 0,C 180,E1 -13661.703,E2 -13661.703} C_VEL
LIN {X 0,Y 319.801,Z 340.408,A -85,B 0,C 180,E1 -13664.402,E2 -13664.402} C_VEL
LIN {X 0,Y 314.261,Z 327.976,A -85,B 0,C 180,E1 -13667.318,E2 -13667.318} C_VEL
LIN {X 0,Y 309.222,Z 318.517,A -85,B 0,C 180,E1 -13669.944,E2 -13669.944} C_VEL
LIN {X 0,Y 306.971,Z 314.379,A -85,B 0,C 180,E1 -13671.193,E2 -13671.193} C_VEL
LIN {X 0,Y 304.436,Z 309.854,A -85,B 0,C 180,E1 -13672.64,E2 -13672.64} C_VEL
LIN {X 0,Y 302.17,Z 306.458,A -85,B 0,C 180,E1 -13673.921,E2 -13673.921} C_VEL
LIN {X 0,Y 301.328,Z 304.672,A -85,B 0,C 180,E1 -13674.504,E2 -13674.504} C_VEL
LIN {X 0,Y 299.045,Z 301.904,A -85,B 0,C 180,E1 -13675.781,E2 -13675.781} C_VEL
LIN {X 0,Y 298.345,Z 299.72,A -85,B 0,C 180,E1 -13676.541,E2 -13676.541} C_VEL
LIN {X 0,Y 298.266,Z 299.329,A -85,B 0,C 180,E1 -13677.694,E2 -13677.694} C_VEL
LIN {X 0,Y 298.272,Z 299.329,A -85,B 0,C 180,E1 -13682.113,E2 -13682.113} C_VEL
LIN {X 0,Y 298.3,Z 299.319,A -85,B 0,C 180,E1 -13686.737,E2 -13686.737} C_VEL
LIN {X 0,Y 298.284,Z 299.331,A -85,B 0,C 180,E1 -13691.21,E2 -13691.21} C_VEL
LIN {X 0,Y 298.27,Z 299.322,A -85,B 0,C 180,E1 -13695.84,E2 -13695.84} C_VEL
LIN {X 0,Y 298.281,Z 299.332,A -85,B 0,C 180,E1 -13700.402,E2 -13700.402} C_VEL
LIN {X 0,Y 298.292,Z 299.323,A -85,B 0,C 180,E1 -13704.77,E2 -13704.77} C_VEL
LIN {X 0,Y 298.325,Z 299.565,A -85,B 0,C 180,E1 -13708.59,E2 -13708.59} C_VEL
LIN {X 0,Y 301.597,Z 307.018,A -85,B 0,C 180,E1 -13710.699,E2 -13710.699} C_VEL
LIN {X 0,Y 307.776,Z 320.683,A -85,B 0,C 180,E1 -13714.195,E2 -13714.195} C_VEL
LIN {X 0,Y 309.708,Z 324.106,A -85,B 0,C 180,E1 -13714.821,E2 -13714.821} C_VEL
LIN {X 0,Y 322.915,Z 345.738,A -85,B 0,C 180,E1 -13717.896,E2 -13717.896} C_VEL
LIN {X 0,Y 337.2,Z 370.561,A -85,B 0,C 180,E1 -13720.942,E2 -13720.942} C_VEL
LIN {X 0,Y 343.751,Z 382.926,A -85,B 0,C 180,E1 -13722.265,E2 -13722.265} C_VEL
LIN {X 0,Y 330.104,Z 576.48,A -85,B 0,C 180,E1 -13727.566,E2 -13727.566} C_VEL
LIN {X 0,Y 327.862,Z 597.383,A -85,B 0,C 180,E1 -13728.424,E2 -13728.424} C_VEL
LIN {X 0,Y 324.939,Z 618.799,A -85,B 0,C 180,E1 -13729.633,E2 -13729.633} C_VEL
LIN {X 0,Y 321.68,Z 638.915,A -85,B 0,C 180,E1 -13731.11,E2 -13731.11} C_VEL
LIN {X 0,Y 318.143,Z 658.191,A -85,B 0,C 180,E1 -13732.888,E2 -13732.888} C_VEL
LIN {X 0,Y 314.434,Z 676.579,A -85,B 0,C 180,E1 -13734.976,E2 -13734.976} C_VEL
LIN {X 0,Y 310.714,Z 693.994,A -85,B 0,C 180,E1 -13737.387,E2 -13737.387} C_VEL
LIN {X 0,Y 307.104,Z 710.311,A -85,B 0,C 180,E1 -13740.126,E2 -13740.126} C_VEL
LIN {X 0,Y 303.92,Z 724.797,A -85,B 0,C 180,E1 -13743.068,E2 -13743.068} C_VEL
LIN {X 0,Y 301.149,Z 738,A -85,B 0,C 180,E1 -13746.316,E2 -13746.316} C_VEL
LIN {X 0,Y 299.039,Z 749.118,A -85,B 0,C 180,E1 -13749.654,E2 -13749.654} C_VEL
LIN {X 0,Y 297.581,Z 758.21,A -85,B 0,C 180,E1 -13753.006,E2 -13753.006} C_VEL
LIN {X 0,Y 296.642,Z 765.905,A -85,B 0,C 180,E1 -13756.554,E2 -13756.554} C_VEL
LIN {X 0,Y 296.206,Z 772.062,A -85,B 0,C 180,E1 -13760.286,E2 -13760.286} C_VEL
LIN {X 0,Y 296.13,Z 776.162,A -85,B 0,C 180,E1 -13763.8,E2 -13763.8} C_VEL
LIN {X 0,Y 296.158,Z 778.504,A -85,B 0,C 180,E1 -13767.099,E2 -13767.099} C_VEL
LIN {X 0,Y 296.169,Z 779.439,A -85,B 0,C 180,E1 -13770.582,E2 -13770.582} C_VEL
LIN {X 0,Y 296.093,Z 778.868,A -85,B 0,C 180,E1 -13774.069,E2 -13774.069} C_VEL
LIN {X 0,Y 296.058,Z 776.743,A -85,B 0,C 180,E1 -13777.571,E2 -13777.571} C_VEL
LIN {X 0,Y 296.292,Z 772.837,A -85,B 0,C 180,E1 -13781.289,E2 -13781.289} C_VEL
LIN {X 0,Y 297.09,Z 766.881,A -85,B 0,C 180,E1 -13785.221,E2 -13785.221} C_VEL
LIN {X 0,Y 298.686,Z 758.943,A -85,B 0,C 180,E1 -13789.153,E2 -13789.153} C_VEL
LIN {X 0,Y 301.255,Z 748.864,A -85,B 0,C 180,E1 -13793.058,E2 -13793.058} C_VEL
LIN {X 0,Y 304.703,Z 737.116,A -85,B 0,C 180,E1 -13796.717,E2 -13796.717} C_VEL
LIN {X 0,Y 308.962,Z 723.842,A -85,B 0,C 180,E1 -13800.108,E2 -13800.108} C_VEL
LIN {X 0,Y 313.936,Z 709.114,A -85,B 0,C 180,E1 -13803.218,E2 -13803.218} C_VEL
LIN {X 0,Y 320.074,Z 691.451,A -85,B 0,C 180,E1 -13806.299,E2 -13806.299} C_VEL
LIN {X 0,Y 326.902,Z 672.158,A -85,B 0,C 180,E1 -13809.057,E2 -13809.057} C_VEL
LIN {X 0,Y 334.096,Z 652.043,A -85,B 0,C 180,E1 -13811.408,E2 -13811.408} C_VEL
LIN {X 0,Y 341.77,Z 630.618,A -85,B 0,C 180,E1 -13813.434,E2 -13813.434} C_VEL
LIN {X 0,Y 349.239,Z 609.57,A -85,B 0,C 180,E1 -13815.005,E2 -13815.005} C_VEL
LIN {X 0,Y 356.52,Z 588.153,A -85,B 0,C 180,E1 -13816.235,E2 -13816.235} C_VEL
LIN {X 0,Y 362.999,Z 567.158,A -85,B 0,C 180,E1 -13817.152,E2 -13817.152} C_VEL
LIN {X 0,Y 356.075,Z 588.45,A -85,B 0,C 180,E1 -13818.172,E2 -13818.172} C_VEL
LIN {X 0,Y 348.708,Z 608.687,A -85,B 0,C 180,E1 -13819.501,E2 -13819.501} C_VEL
LIN {X 0,Y 340.907,Z 628.961,A -85,B 0,C 180,E1 -13821.232,E2 -13821.232} C_VEL
LIN {X 0,Y 333.005,Z 649.1,A -85,B 0,C 180,E1 -13823.416,E2 -13823.416} C_VEL
LIN {X 0,Y 325.721,Z 667.773,A -85,B 0,C 180,E1 -13825.93,E2 -13825.93} C_VEL
LIN {X 0,Y 319.256,Z 684.33,A -85,B 0,C 180,E1 -13828.676,E2 -13828.676} C_VEL
LIN {X 0,Y 313.526,Z 699.018,A -85,B 0,C 180,E1 -13831.667,E2 -13831.667} C_VEL
LIN {X 0,Y 308.596,Z 711.853,A -85,B 0,C 180,E1 -13834.885,E2 -13834.885} C_VEL
LIN {X 0,Y 304.585,Z 722.584,A -85,B 0,C 180,E1 -13838.227,E2 -13838.227} C_VEL
LIN {X 0,Y 301.485,Z 731.267,A -85,B 0,C 180,E1 -13841.636,E2 -13841.636} C_VEL
LIN {X 0,Y 299.226,Z 738.076,A -85,B 0,C 180,E1 -13845.091,E2 -13845.091} C_VEL
LIN {X 0,Y 297.712,Z 743.131,A -85,B 0,C 180,E1 -13848.572,E2 -13848.572} C_VEL
LIN {X 0,Y 296.799,Z 746.534,A -85,B 0,C 180,E1 -13852.076,E2 -13852.076} C_VEL
LIN {X 0,Y 296.337,Z 748.357,A -85,B 0,C 180,E1 -13855.744,E2 -13855.744} C_VEL
LIN {X 0,Y 296.181,Z 748.441,A -85,B 0,C 180,E1 -13859.227,E2 -13859.227} C_VEL
LIN {X 0,Y 296.143,Z 746.897,A -85,B 0,C 180,E1 -13862.71,E2 -13862.71} C_VEL
LIN {X 0,Y 296.246,Z 743.918,A -85,B 0,C 180,E1 -13866.006,E2 -13866.006} C_VEL
LIN {X 0,Y 296.583,Z 739.38,A -85,B 0,C 180,E1 -13869.313,E2 -13869.313} C_VEL
LIN {X 0,Y 297.345,Z 732.714,A -85,B 0,C 180,E1 -13872.823,E2 -13872.823} C_VEL
LIN {X 0,Y 298.573,Z 724.542,A -85,B 0,C 180,E1 -13876.139,E2 -13876.139} C_VEL
LIN {X 0,Y 300.398,Z 714.286,A -85,B 0,C 180,E1 -13879.442,E2 -13879.442} C_VEL
LIN {X 0,Y 302.724,Z 702.453,A -85,B 0,C 180,E1 -13882.529,E2 -13882.529} C_VEL
LIN {X 0,Y 305.487,Z 689.043,A -85,B 0,C 180,E1 -13885.395,E2 -13885.395} C_VEL
LIN {X 0,Y 308.576,Z 674.094,A -85,B 0,C 180,E1 -13888.024,E2 -13888.024} C_VEL
LIN {X 0,Y 311.911,Z 657.424,A -85,B 0,C 180,E1 -13890.431,E2 -13890.431} C_VEL
LIN {X 0,Y 315.11,Z 640.48,A -85,B 0,C 180,E1 -13892.429,E2 -13892.429} C_VEL
LIN {X 0,Y 318.315,Z 621.836,A -85,B 0,C 180,E1 -13894.213,E2 -13894.213} C_VEL
LIN {X 0,Y 321.259,Z 602.305,A -85,B 0,C 180,E1 -13895.691,E2 -13895.691} C_VEL
LIN {X 0,Y 323.833,Z 581.753,A -85,B 0,C 180,E1 -13896.868,E2 -13896.868} C_VEL
LIN {X 0,Y 325.84,Z 561.087,A -85,B 0,C 180,E1 -13897.713,E2 -13897.713} C_VEL
LIN {X 0,Y 338.284,Z 387.696,A -85,B 0,C 180,E1 -13902.711,E2 -13902.711} C_VEL
LIN {X 0,Y 337.288,Z 380.441,A -85,B 0,C 180,E1 -13903.113,E2 -13903.113} C_VEL
LIN {X 0,Y 324.016,Z 355.169,A -85,B 0,C 180,E1 -13905.934,E2 -13905.934} C_VEL
LIN {X 0,Y 314.242,Z 337.598,A -85,B 0,C 180,E1 -13908.194,E2 -13908.194} C_VEL
LIN {X 0,Y 307.561,Z 321.152,A -85,B 0,C 180,E1 -13912.088,E2 -13912.088} C_VEL
LIN {X 0,Y 301.696,Z 307.291,A -85,B 0,C 180,E1 -13915.707,E2 -13915.707} C_VEL
LIN {X 0,Y 298.35,Z 299.669,A -85,B 0,C 180,E1 -13917.913,E2 -13917.913} C_VEL
LIN {X 0,Y 298.344,Z 299.647,A -85,B 0,C 180,E1 -13918.349,E2 -13918.349} C_VEL
LIN {X 0,Y 299.473,Z 302.618,A -85,B 0,C 180,E1 -13919.1,E2 -13919.1} C_VEL
LIN {X 0,Y 300.763,Z 304.67,A -85,B 0,C 180,E1 -13919.646,E2 -13919.646} C_VEL
LIN {X 0,Y 307.285,Z 317.966,A -85,B 0,C 180,E1 -13922.689,E2 -13922.689} C_VEL
LIN {X 0,Y 313.789,Z 332.45,A -85,B 0,C 180,E1 -13925.689,E2 -13925.689} C_VEL
LIN {X 0,Y 320.234,Z 349.04,A -85,B 0,C 180,E1 -13928.764,E2 -13928.764} C_VEL
LIN {X 0,Y 325.746,Z 365.749,A -85,B 0,C 180,E1 -13931.568,E2 -13931.568} C_VEL
LIN {X 0,Y 326.196,Z 367.588,A -85,B 0,C 180,E1 -13931.847,E2 -13931.847} C_VEL
LIN {X 0,Y 322.078,Z 408.691,A -85,B 0,C 180,E1 -13936.168,E2 -13936.168} C_VEL
LIN {X 0,Y 318.024,Z 450.872,A -85,B 0,C 180,E1 -13940.589,E2 -13940.589} C_VEL
LIN {X 0,Y 315.078,Z 483.048,A -85,B 0,C 180,E1 -13943.953,E2 -13943.953} C_VEL
LIN {X 0,Y 317.125,Z 505.823,A -85,B 0,C 180,E1 -13944.758,E2 -13944.758} C_VEL
LIN {X 0,Y 313.15,Z 627.003,A -85,B 0,C 180,E1 -13947.573,E2 -13947.573} C_VEL
LIN {X 0,Y 312.156,Z 643.081,A -85,B 0,C 180,E1 -13948.279,E2 -13948.279} C_VEL
LIN {X 0,Y 310.63,Z 659.442,A -85,B 0,C 180,E1 -13949.353,E2 -13949.353} C_VEL
LIN {X 0,Y 308.843,Z 673.77,A -85,B 0,C 180,E1 -13950.647,E2 -13950.647} C_VEL
LIN {X 0,Y 306.706,Z 688.146,A -85,B 0,C 180,E1 -13952.333,E2 -13952.333} C_VEL
LIN {X 0,Y 305.895,Z 693.038,A -85,B 0,C 180,E1 -13953.018,E2 -13953.018} C_VEL
LIN {X 0,Y 303.942,Z 699.059,A -85,B 0,C 180,E1 -13953.864,E2 -13953.864} C_VEL
LIN {X 0,Y 297.366,Z 710.104,A -85,B 0,C 180,E1 -13955.572,E2 -13955.572} C_VEL
LIN {X 0,Y 294.321,Z 715.969,A -85,B 0,C 180,E1 -13956.729,E2 -13956.729} C_VEL
LIN {X 0,Y 293.713,Z 718.085,A -85,B 0,C 180,E1 -13957.216,E2 -13957.216} C_VEL
LIN {X 0,Y 291.804,Z 727.607,A -85,B 0,C 180,E1 -13959.863,E2 -13959.863} C_VEL
LIN {X 0,Y 290.267,Z 735.655,A -85,B 0,C 180,E1 -13962.733,E2 -13962.733} C_VEL
LIN {X 0,Y 289.154,Z 742.088,A -85,B 0,C 180,E1 -13965.851,E2 -13965.851} C_VEL
LIN {X 0,Y 288.521,Z 746.641,A -85,B 0,C 180,E1 -13969.009,E2 -13969.009} C_VEL
LIN {X 0,Y 288.245,Z 749.351,A -85,B 0,C 180,E1 -13972.213,E2 -13972.213} C_VEL
LIN {X 0,Y 288.194,Z 750.361,A -85,B 0,C 180,E1 -13975.478,E2 -13975.478} C_VEL
LIN {X 0,Y 288.325,Z 749.547,A -85,B 0,C 180,E1 -13978.673,E2 -13978.673} C_VEL
LIN {X 0,Y 288.758,Z 746.923,A -85,B 0,C 180,E1 -13981.988,E2 -13981.988} C_VEL
LIN {X 0,Y 289.613,Z 742.414,A -85,B 0,C 180,E1 -13985.205,E2 -13985.205} C_VEL
LIN {X 0,Y 290.942,Z 736.368,A -85,B 0,C 180,E1 -13988.21,E2 -13988.21} C_VEL
LIN {X 0,Y 292.684,Z 728.836,A -85,B 0,C 180,E1 -13990.985,E2 -13990.985} C_VEL
LIN {X 0,Y 294.971,Z 719.136,A -85,B 0,C 180,E1 -13993.745,E2 -13993.745} C_VEL
LIN {X 0,Y 297.299,Z 708.873,A -85,B 0,C 180,E1 -13996.027,E2 -13996.027} C_VEL
LIN {X 0,Y 299.864,Z 696.725,A -85,B 0,C 180,E1 -13998.173,E2 -13998.173} C_VEL
LIN {X 0,Y 302.288,Z 683.918,A -85,B 0,C 180,E1 -13999.959,E2 -13999.959} C_VEL
LIN {X 0,Y 304.649,Z 669.338,A -85,B 0,C 180,E1 -14001.534,E2 -14001.534} C_VEL
LIN {X 0,Y 306.551,Z 654.728,A -85,B 0,C 180,E1 -14002.73,E2 -14002.73} C_VEL
LIN {X 0,Y 308.074,Z 638.124,A -85,B 0,C 180,E1 -14003.693,E2 -14003.693} C_VEL
LIN {X 0,Y 308.979,Z 621.885,A -85,B 0,C 180,E1 -14004.284,E2 -14004.284} C_VEL
LIN {X 0,Y 313.276,Z 504.516,A -85,B 0,C 180,E1 -14007.076,E2 -14007.076} C_VEL
LIN {X 0,Y 311.269,Z 483.706,A -85,B 0,C 180,E1 -14007.993,E2 -14007.993} C_VEL
LIN {X 0,Y 315.775,Z 440.448,A -85,B 0,C 180,E1 -14012.566,E2 -14012.566} C_VEL
LIN {X 0,Y 320.259,Z 399.816,A -85,B 0,C 180,E1 -14016.835,E2 -14016.835} C_VEL
LIN {X 0,Y 323.216,Z 372.036,A -85,B 0,C 180,E1 -14019.728,E2 -14019.728} C_VEL
LIN {X 0,Y 318.951,Z 357.97,A -85,B 0,C 180,E1 -14022.296,E2 -14022.296} C_VEL
LIN {X 0,Y 314.031,Z 344.867,A -85,B 0,C 180,E1 -14025.054,E2 -14025.054} C_VEL
LIN {X 0,Y 308.721,Z 332.948,A -85,B 0,C 180,E1 -14027.971,E2 -14027.971} C_VEL
LIN {X 0,Y 304.464,Z 324.564,A -85,B 0,C 180,E1 -14030.358,E2 -14030.358} C_VEL
LIN {X 0,Y 301.878,Z 319.942,A -85,B 0,C 180,E1 -14031.811,E2 -14031.811} C_VEL
LIN {X 0,Y 299.851,Z 316.089,A -85,B 0,C 180,E1 -14033.105,E2 -14033.105} C_VEL
LIN {X 0,Y 297.685,Z 312.569,A -85,B 0,C 180,E1 -14034.41,E2 -14034.41} C_VEL
LIN {X 0,Y 296.81,Z 311.061,A -85,B 0,C 180,E1 -14034.975,E2 -14034.975} C_VEL
LIN {X 0,Y 294.525,Z 307.738,A -85,B 0,C 180,E1 -14036.4,E2 -14036.4} C_VEL
LIN {X 0,Y 293.685,Z 305.893,A -85,B 0,C 180,E1 -14037.072,E2 -14037.072} C_VEL
LIN {X 0,Y 291.271,Z 303.159,A -85,B 0,C 180,E1 -14038.622,E2 -14038.622} C_VEL
LIN {X 0,Y 290.382,Z 300.676,A -85,B 0,C 180,E1 -14039.703,E2 -14039.703} C_VEL
LIN {X 0,Y 290.33,Z 300.314,A -85,B 0,C 180,E1 -14041.578,E2 -14041.578} C_VEL
LIN {X 0,Y 290.341,Z 300.312,A -85,B 0,C 180,E1 -14046.326,E2 -14046.326} C_VEL
LIN {X 0,Y 290.352,Z 300.315,A -85,B 0,C 180,E1 -14050.917,E2 -14050.917} C_VEL
LIN {X 0,Y 290.337,Z 300.31,A -85,B 0,C 180,E1 -14055.581,E2 -14055.581} C_VEL
LIN {X 0,Y 290.341,Z 300.32,A -85,B 0,C 180,E1 -14060.353,E2 -14060.353} C_VEL
LIN {X 0,Y 290.353,Z 300.311,A -85,B 0,C 180,E1 -14064.841,E2 -14064.841} C_VEL
LIN {X 0,Y 290.4,Z 300.603,A -85,B 0,C 180,E1 -14067.102,E2 -14067.102} C_VEL
LIN {X 0,Y 291.95,Z 304.252,A -85,B 0,C 180,E1 -14068.204,E2 -14068.204} C_VEL
LIN {X 0,Y 297.957,Z 317.252,A -85,B 0,C 180,E1 -14071.792,E2 -14071.792} C_VEL
LIN {X 0,Y 300.495,Z 322.749,A -85,B 0,C 180,E1 -14073.128,E2 -14073.128} C_VEL
LIN {X 0,Y 312.992,Z 342.953,A -85,B 0,C 180,E1 -14076.226,E2 -14076.226} C_VEL
LIN {X 0,Y 326.944,Z 366.814,A -85,B 0,C 180,E1 -14079.36,E2 -14079.36} C_VEL
LIN {X 0,Y 337.203,Z 385.814,A -85,B 0,C 180,E1 -14081.515,E2 -14081.515} C_VEL
LIN {X 0,Y 323.152,Z 576.47,A -85,B 0,C 180,E1 -14086.871,E2 -14086.871} C_VEL
LIN {X 0,Y 320.716,Z 598.189,A -85,B 0,C 180,E1 -14087.794,E2 -14087.794} C_VEL
LIN {X 0,Y 317.763,Z 619.003,A -85,B 0,C 180,E1 -14089.004,E2 -14089.004} C_VEL
LIN {X 0,Y 314.412,Z 638.998,A -85,B 0,C 180,E1 -14090.508,E2 -14090.508} C_VEL
LIN {X 0,Y 310.637,Z 658.851,A -85,B 0,C 180,E1 -14092.391,E2 -14092.391} C_VEL
LIN {X 0,Y 306.793,Z 677.253,A -85,B 0,C 180,E1 -14094.544,E2 -14094.544} C_VEL
LIN {X 0,Y 302.977,Z 694.529,A -85,B 0,C 180,E1 -14097.011,E2 -14097.011} C_VEL
LIN {X 0,Y 299.277,Z 710.724,A -85,B 0,C 180,E1 -14099.817,E2 -14099.817} C_VEL
LIN {X 0,Y 295.977,Z 725.269,A -85,B 0,C 180,E1 -14102.87,E2 -14102.87} C_VEL
LIN {X 0,Y 293.253,Z 737.871,A -85,B 0,C 180,E1 -14106.065,E2 -14106.065} C_VEL
LIN {X 0,Y 291.083,Z 748.968,A -85,B 0,C 180,E1 -14109.493,E2 -14109.493} C_VEL
LIN {X 0,Y 289.556,Z 758.27,A -85,B 0,C 180,E1 -14113.037,E2 -14113.037} C_VEL
LIN {X 0,Y 288.64,Z 765.677,A -85,B 0,C 180,E1 -14116.582,E2 -14116.582} C_VEL
LIN {X 0,Y 288.223,Z 771.51,A -85,B 0,C 180,E1 -14120.215,E2 -14120.215} C_VEL
LIN {X 0,Y 288.147,Z 775.657,A -85,B 0,C 180,E1 -14123.827,E2 -14123.827} C_VEL
LIN {X 0,Y 288.179,Z 777.998,A -85,B 0,C 180,E1 -14127.218,E2 -14127.218} C_VEL
LIN {X 0,Y 288.182,Z 778.943,A -85,B 0,C 180,E1 -14130.797,E2 -14130.797} C_VEL
LIN {X 0,Y 288.097,Z 778.471,A -85,B 0,C 180,E1 -14134.182,E2 -14134.182} C_VEL
LIN {X 0,Y 288.066,Z 776.393,A -85,B 0,C 180,E1 -14137.782,E2 -14137.782} C_VEL
LIN {X 0,Y 288.327,Z 772.596,A -85,B 0,C 180,E1 -14141.605,E2 -14141.605} C_VEL
LIN {X 0,Y 289.217,Z 766.77,A -85,B 0,C 180,E1 -14145.646,E2 -14145.646} C_VEL
LIN {X 0,Y 290.858,Z 759.44,A -85,B 0,C 180,E1 -14149.48,E2 -14149.48} C_VEL
LIN {X 0,Y 293.432,Z 750.237,A -85,B 0,C 180,E1 -14153.285,E2 -14153.285} C_VEL
LIN {X 0,Y 297.038,Z 738.999,A -85,B 0,C 180,E1 -14157.03,E2 -14157.03} C_VEL
LIN {X 0,Y 301.763,Z 725.517,A -85,B 0,C 180,E1 -14160.683,E2 -14160.683} C_VEL
LIN {X 0,Y 307.353,Z 710.484,A -85,B 0,C 180,E1 -14164.026,E2 -14164.026} C_VEL
LIN {X 0,Y 313.874,Z 693.503,A -85,B 0,C 180,E1 -14167.134,E2 -14167.134} C_VEL
LIN {X 0,Y 321.336,Z 674.56,A -85,B 0,C 180,E1 -14169.983,E2 -14169.983} C_VEL
LIN {X 0,Y 329.771,Z 653.621,A -85,B 0,C 180,E1 -14172.544,E2 -14172.544} C_VEL
LIN {X 0,Y 338.598,Z 632.089,A -85,B 0,C 180,E1 -14174.654,E2 -14174.654} C_VEL
LIN {X 0,Y 346.932,Z 611.698,A -85,B 0,C 180,E1 -14176.217,E2 -14176.217} C_VEL
LIN {X 0,Y 353.303,Z 595.395,A -85,B 0,C 180,E1 -14177.219,E2 -14177.219} C_VEL
LIN {X 0,Y 345.191,Z 614.593,A -85,B 0,C 180,E1 -14178.559,E2 -14178.559} C_VEL
LIN {X 0,Y 336.339,Z 634.602,A -85,B 0,C 180,E1 -14180.383,E2 -14180.383} C_VEL
LIN {X 0,Y 327.74,Z 653.944,A -85,B 0,C 180,E1 -14182.62,E2 -14182.62} C_VEL
LIN {X 0,Y 319.55,Z 672.365,A -85,B 0,C 180,E1 -14185.287,E2 -14185.287} C_VEL
LIN {X 0,Y 312.175,Z 689.25,A -85,B 0,C 180,E1 -14188.314,E2 -14188.314} C_VEL
LIN {X 0,Y 306.281,Z 702.933,A -85,B 0,C 180,E1 -14191.323,E2 -14191.323} C_VEL
LIN {X 0,Y 301.089,Z 715.166,A -85,B 0,C 180,E1 -14194.636,E2 -14194.636} C_VEL
LIN {X 0,Y 296.9,Z 725.271,A -85,B 0,C 180,E1 -14198.05,E2 -14198.05} C_VEL
LIN {X 0,Y 293.669,Z 733.454,A -85,B 0,C 180,E1 -14201.541,E2 -14201.541} C_VEL
LIN {X 0,Y 291.208,Z 740.129,A -85,B 0,C 180,E1 -14205.282,E2 -14205.282} C_VEL
LIN {X 0,Y 289.609,Z 744.92,A -85,B 0,C 180,E1 -14209.055,E2 -14209.055} C_VEL
LIN {X 0,Y 288.741,Z 747.807,A -85,B 0,C 180,E1 -14212.639,E2 -14212.639} C_VEL
LIN {X 0,Y 288.328,Z 749.088,A -85,B 0,C 180,E1 -14216.223,E2 -14216.223} C_VEL
LIN {X 0,Y 288.179,Z 748.739,A -85,B 0,C 180,E1 -14219.802,E2 -14219.802} C_VEL
LIN {X 0,Y 288.157,Z 746.816,A -85,B 0,C 180,E1 -14223.305,E2 -14223.305} C_VEL
LIN {X 0,Y 288.3,Z 743.34,A -85,B 0,C 180,E1 -14226.773,E2 -14226.773} C_VEL
LIN {X 0,Y 288.728,Z 738.333,A -85,B 0,C 180,E1 -14230.173,E2 -14230.173} C_VEL
LIN {X 0,Y 289.635,Z 731.172,A -85,B 0,C 180,E1 -14233.781,E2 -14233.781} C_VEL
LIN {X 0,Y 291.102,Z 722.203,A -85,B 0,C 180,E1 -14237.277,E2 -14237.277} C_VEL
LIN {X 0,Y 293.114,Z 711.618,A -85,B 0,C 180,E1 -14240.571,E2 -14240.571} C_VEL
LIN {X 0,Y 295.699,Z 699.133,A -85,B 0,C 180,E1 -14243.728,E2 -14243.728} C_VEL
LIN {X 0,Y 298.744,Z 684.919,A -85,B 0,C 180,E1 -14246.666,E2 -14246.666} C_VEL
LIN {X 0,Y 302.094,Z 669.098,A -85,B 0,C 180,E1 -14249.331,E2 -14249.331} C_VEL
LIN {X 0,Y 305.413,Z 652.778,A -85,B 0,C 180,E1 -14251.589,E2 -14251.589} C_VEL
LIN {X 0,Y 308.822,Z 634.784,A -85,B 0,C 180,E1 -14253.618,E2 -14253.618} C_VEL
LIN {X 0,Y 312.045,Z 615.813,A -85,B 0,C 180,E1 -14255.336,E2 -14255.336} C_VEL
LIN {X 0,Y 314.995,Z 595.834,A -85,B 0,C 180,E1 -14256.752,E2 -14256.752} C_VEL
LIN {X 0,Y 317.501,Z 575.057,A -85,B 0,C 180,E1 -14257.858,E2 -14257.858} C_VEL
LIN {X 0,Y 319.444,Z 553.628,A -85,B 0,C 180,E1 -14258.649,E2 -14258.649} C_VEL
LIN {X 0,Y 331.795,Z 388.835,A -85,B 0,C 180,E1 -14263.504,E2 -14263.504} C_VEL
LIN {X 0,Y 331.062,Z 383.919,A -85,B 0,C 180,E1 -14263.793,E2 -14263.793} C_VEL
LIN {X 0,Y 317.662,Z 358.305,A -85,B 0,C 180,E1 -14266.733,E2 -14266.733} C_VEL
LIN {X 0,Y 305.918,Z 337.309,A -85,B 0,C 180,E1 -14269.561,E2 -14269.561} C_VEL
LIN {X 0,Y 299.661,Z 322.098,A -85,B 0,C 180,E1 -14273.324,E2 -14273.324} C_VEL
LIN {X 0,Y 293.724,Z 308.207,A -85,B 0,C 180,E1 -14277.113,E2 -14277.113} C_VEL
LIN {X 0,Y 292.649,Z 305.817,A -85,B 0,C 180,E1 -14277.922,E2 -14277.922} C_VEL
LIN {X 0,Y 292.995,Z 305.922,A -85,B 0,C 180,E1 -14278.183,E2 -14278.183} C_VEL
LIN {X 0,Y 299.337,Z 318.491,A -85,B 0,C 180,E1 -14281.248,E2 -14281.248} C_VEL
LIN {X 0,Y 305.719,Z 332.398,A -85,B 0,C 180,E1 -14284.295,E2 -14284.295} C_VEL
LIN {X 0,Y 312.314,Z 348.839,A -85,B 0,C 180,E1 -14287.515,E2 -14287.515} C_VEL
LIN {X 0,Y 317.97,Z 365.473,A -85,B 0,C 180,E1 -14290.432,E2 -14290.432} C_VEL
LIN {X 0,Y 319.369,Z 370.759,A -85,B 0,C 180,E1 -14291.281,E2 -14291.281} C_VEL
LIN {X 0,Y 315.086,Z 412.181,A -85,B 0,C 180,E1 -14295.668,E2 -14295.668} C_VEL
LIN {X 0,Y 310.52,Z 457.184,A -85,B 0,C 180,E1 -14300.453,E2 -14300.453} C_VEL
LIN {X 0,Y 308.06,Z 483.467,A -85,B 0,C 180,E1 -14303.226,E2 -14303.226} C_VEL
LIN {X 0,Y 310.09,Z 506.695,A -85,B 0,C 180,E1 -14304.07,E2 -14304.07} C_VEL
LIN {X 0,Y 305.942,Z 627.479,A -85,B 0,C 180,E1 -14306.936,E2 -14306.936} C_VEL
LIN {X 0,Y 304.89,Z 643.68,A -85,B 0,C 180,E1 -14307.666,E2 -14307.666} C_VEL
LIN {X 0,Y 303.423,Z 658.854,A -85,B 0,C 180,E1 -14308.676,E2 -14308.676} C_VEL
LIN {X 0,Y 301.562,Z 673.458,A -85,B 0,C 180,E1 -14309.998,E2 -14309.998} C_VEL
LIN {X 0,Y 299.322,Z 687.963,A -85,B 0,C 180,E1 -14311.721,E2 -14311.721} C_VEL
LIN {X 0,Y 297.06,Z 700.729,A -85,B 0,C 180,E1 -14313.664,E2 -14313.664} C_VEL
LIN {X 0,Y 294.728,Z 712.976,A -85,B 0,C 180,E1 -14316.035,E2 -14316.035} C_VEL
LIN {X 0,Y 293.713,Z 718.085,A -85,B 0,C 180,E1 -14317.216,E2 -14317.216} C_VEL
LIN {X 0,Y 291.83,Z 722.819,A -85,B 0,C 180,E1 -14318.365,E2 -14318.365} C_VEL
LIN {X 0,Y 285.957,Z 730.646,A -85,B 0,C 180,E1 -14320.503,E2 -14320.503} C_VEL
LIN {X 0,Y 282.972,Z 734.859,A -85,B 0,C 180,E1 -14321.97,E2 -14321.97} C_VEL
LIN {X 0,Y 282.245,Z 736.774,A -85,B 0,C 180,E1 -14322.77,E2 -14322.77} C_VEL
LIN {X 0,Y 281.151,Z 742.896,A -85,B 0,C 180,E1 -14325.89,E2 -14325.89} C_VEL
LIN {X 0,Y 280.543,Z 747.061,A -85,B 0,C 180,E1 -14328.922,E2 -14328.922} C_VEL
LIN {X 0,Y 280.254,Z 749.76,A -85,B 0,C 180,E1 -14332.218,E2 -14332.218} C_VEL
LIN {X 0,Y 280.205,Z 750.754,A -85,B 0,C 180,E1 -14335.577,E2 -14335.577} C_VEL
LIN {X 0,Y 280.346,Z 749.97,A -85,B 0,C 180,E1 -14338.779,E2 -14338.779} C_VEL
LIN {X 0,Y 280.786,Z 747.499,A -85,B 0,C 180,E1 -14342.058,E2 -14342.058} C_VEL
LIN {X 0,Y 281.65,Z 743.296,A -85,B 0,C 180,E1 -14345.262,E2 -14345.262} C_VEL
LIN {X 0,Y 283.066,Z 737.211,A -85,B 0,C 180,E1 -14348.435,E2 -14348.435} C_VEL
LIN {X 0,Y 284.919,Z 729.728,A -85,B 0,C 180,E1 -14351.323,E2 -14351.323} C_VEL
LIN {X 0,Y 287.365,Z 719.911,A -85,B 0,C 180,E1 -14354.211,E2 -14354.211} C_VEL
LIN {X 0,Y 289.96,Z 709.115,A -85,B 0,C 180,E1 -14356.68,E2 -14356.68} C_VEL
LIN {X 0,Y 292.694,Z 696.846,A -85,B 0,C 180,E1 -14358.89,E2 -14358.89} C_VEL
LIN {X 0,Y 295.237,Z 684.023,A -85,B 0,C 180,E1 -14360.705,E2 -14360.705} C_VEL
LIN {X 0,Y 297.737,Z 669.235,A -85,B 0,C 180,E1 -14362.323,E2 -14362.323} C_VEL
LIN {X 0,Y 299.684,Z 654.782,A -85,B 0,C 180,E1 -14363.516,E2 -14363.516} C_VEL
LIN {X 0,Y 301.286,Z 637.985,A -85,B 0,C 180,E1 -14364.498,E2 -14364.498} C_VEL
LIN {X 0,Y 302.215,Z 621.596,A -85,B 0,C 180,E1 -14365.092,E2 -14365.092} C_VEL
LIN {X 0,Y 306.717,Z 505.397,A -85,B 0,C 180,E1 -14367.915,E2 -14367.915} C_VEL
LIN {X 0,Y 304.744,Z 483.938,A -85,B 0,C 180,E1 -14368.902,E2 -14368.902} C_VEL
LIN {X 0,Y 309.476,Z 440.771,A -85,B 0,C 180,E1 -14373.521,E2 -14373.521} C_VEL
LIN {X 0,Y 313.94,Z 402.011,A -85,B 0,C 180,E1 -14377.629,E2 -14377.629} C_VEL
LIN {X 0,Y 316.94,Z 375.31,A -85,B 0,C 180,E1 -14380.463,E2 -14380.463} C_VEL
LIN {X 0,Y 312.814,Z 361.491,A -85,B 0,C 180,E1 -14383.089,E2 -14383.089} C_VEL
LIN {X 0,Y 308.061,Z 348.584,A -85,B 0,C 180,E1 -14385.911,E2 -14385.911} C_VEL
LIN {X 0,Y 302.482,Z 336.042,A -85,B 0,C 180,E1 -14389.139,E2 -14389.139} C_VEL
LIN {X 0,Y 297.914,Z 327.046,A -85,B 0,C 180,E1 -14391.896,E2 -14391.896} C_VEL
LIN {X 0,Y 295.304,Z 322.305,A -85,B 0,C 180,E1 -14393.584,E2 -14393.584} C_VEL
LIN {X 0,Y 292.649,Z 317.725,A -85,B 0,C 180,E1 -14395.296,E2 -14395.296} C_VEL
LIN {X 0,Y 290.362,Z 314.198,A -85,B 0,C 180,E1 -14396.841,E2 -14396.841} C_VEL
LIN {X 0,Y 289.655,Z 312.683,A -85,B 0,C 180,E1 -14397.427,E2 -14397.427} C_VEL
LIN {X 0,Y 287.148,Z 309.419,A -85,B 0,C 180,E1 -14399.201,E2 -14399.201} C_VEL
LIN {X 0,Y 285.949,Z 307.02,A -85,B 0,C 180,E1 -14400.293,E2 -14400.293} C_VEL
LIN {X 0,Y 283.212,Z 303.942,A -85,B 0,C 180,E1 -14402.488,E2 -14402.488} C_VEL
LIN {X 0,Y 282.445,Z 301.673,A -85,B 0,C 180,E1 -14403.754,E2 -14403.754} C_VEL
LIN {X 0,Y 282.401,Z 301.3,A -85,B 0,C 180,E1 -14406.301,E2 -14406.301} C_VEL
LIN {X 0,Y 282.411,Z 301.306,A -85,B 0,C 180,E1 -14411.021,E2 -14411.021} C_VEL
LIN {X 0,Y 282.397,Z 301.299,A -85,B 0,C 180,E1 -14415.635,E2 -14415.635} C_VEL
LIN {X 0,Y 282.401,Z 301.309,A -85,B 0,C 180,E1 -14420.302,E2 -14420.302} C_VEL
LIN {X 0,Y 282.414,Z 301.3,A -85,B 0,C 180,E1 -14424.916,E2 -14424.916} C_VEL
LIN {X 0,Y 282.492,Z 301.857,A -85,B 0,C 180,E1 -14425.582,E2 -14425.582} C_VEL
LIN {X 0,Y 283.883,Z 305.035,A -85,B 0,C 180,E1 -14426.57,E2 -14426.57} C_VEL
LIN {X 0,Y 288.805,Z 315.63,A -85,B 0,C 180,E1 -14429.674,E2 -14429.674} C_VEL
LIN {X 0,Y 292.298,Z 322.994,A -85,B 0,C 180,E1 -14431.615,E2 -14431.615} C_VEL
LIN {X 0,Y 305.566,Z 344.296,A -85,B 0,C 180,E1 -14435.047,E2 -14435.047} C_VEL
LIN {X 0,Y 319.74,Z 368.482,A -85,B 0,C 180,E1 -14438.369,E2 -14438.369} C_VEL
LIN {X 0,Y 330.685,Z 388.558,A -85,B 0,C 180,E1 -14440.742,E2 -14440.742} C_VEL
LIN {X 0,Y 316.201,Z 576.44,A -85,B 0,C 180,E1 -14446.161,E2 -14446.161} C_VEL
LIN {X 0,Y 313.756,Z 597.587,A -85,B 0,C 180,E1 -14447.075,E2 -14447.075} C_VEL
LIN {X 0,Y 310.649,Z 618.855,A -85,B 0,C 180,E1 -14448.334,E2 -14448.334} C_VEL
LIN {X 0,Y 307.081,Z 639.415,A -85,B 0,C 180,E1 -14449.921,E2 -14449.921} C_VEL
LIN {X 0,Y 303.249,Z 658.915,A -85,B 0,C 180,E1 -14451.817,E2 -14451.817} C_VEL
LIN {X 0,Y 299.33,Z 677.098,A -85,B 0,C 180,E1 -14453.995,E2 -14453.995} C_VEL
LIN {X 0,Y 295.394,Z 694.354,A -85,B 0,C 180,E1 -14456.517,E2 -14456.517} C_VEL
LIN {X 0,Y 291.695,Z 710.039,A -85,B 0,C 180,E1 -14459.29,E2 -14459.29} C_VEL
LIN {X 0,Y 288.371,Z 724.231,A -85,B 0,C 180,E1 -14462.318,E2 -14462.318} C_VEL
LIN {X 0,Y 285.363,Z 737.674,A -85,B 0,C 180,E1 -14465.801,E2 -14465.801} C_VEL
LIN {X 0,Y 283.102,Z 748.923,A -85,B 0,C 180,E1 -14469.377,E2 -14469.377} C_VEL
LIN {X 0,Y 281.531,Z 758.289,A -85,B 0,C 180,E1 -14473.071,E2 -14473.071} C_VEL
LIN {X 0,Y 280.602,Z 765.79,A -85,B 0,C 180,E1 -14476.82,E2 -14476.82} C_VEL
LIN {X 0,Y 280.218,Z 771.466,A -85,B 0,C 180,E1 -14480.555,E2 -14480.555} C_VEL
LIN {X 0,Y 280.161,Z 775.729,A -85,B 0,C 180,E1 -14484.473,E2 -14484.473} C_VEL
LIN {X 0,Y 280.205,Z 777.704,A -85,B 0,C 180,E1 -14487.753,E2 -14487.753} C_VEL
LIN {X 0,Y 280.19,Z 778.447,A -85,B 0,C 180,E1 -14491.229,E2 -14491.229} C_VEL
LIN {X 0,Y 280.083,Z 777.8,A -85,B 0,C 180,E1 -14494.917,E2 -14494.917} C_VEL
LIN {X 0,Y 280.094,Z 775.614,A -85,B 0,C 180,E1 -14498.625,E2 -14498.625} C_VEL
LIN {X 0,Y 280.465,Z 771.646,A -85,B 0,C 180,E1 -14502.562,E2 -14502.562} C_VEL
LIN {X 0,Y 281.59,Z 765.677,A -85,B 0,C 180,E1 -14506.717,E2 -14506.717} C_VEL
LIN {X 0,Y 283.72,Z 757.558,A -85,B 0,C 180,E1 -14510.952,E2 -14510.952} C_VEL
LIN {X 0,Y 287.047,Z 747.253,A -85,B 0,C 180,E1 -14515.15,E2 -14515.15} C_VEL
LIN {X 0,Y 291.557,Z 734.966,A -85,B 0,C 180,E1 -14519.144,E2 -14519.144} C_VEL
LIN {X 0,Y 297.072,Z 721.083,A -85,B 0,C 180,E1 -14522.814,E2 -14522.814} C_VEL
LIN {X 0,Y 303.712,Z 705.238,A -85,B 0,C 180,E1 -14526.239,E2 -14526.239} C_VEL
LIN {X 0,Y 311.353,Z 687.627,A -85,B 0,C 180,E1 -14529.365,E2 -14529.365} C_VEL
LIN {X 0,Y 320.1,Z 668.143,A -85,B 0,C 180,E1 -14532.19,E2 -14532.19} C_VEL
LIN {X 0,Y 329.945,Z 646.738,A -85,B 0,C 180,E1 -14534.674,E2 -14534.674} C_VEL
LIN {X 0,Y 339.525,Z 626.321,A -85,B 0,C 180,E1 -14536.547,E2 -14536.547} C_VEL
LIN {X 0,Y 343.988,Z 616.74,A -85,B 0,C 180,E1 -14537.286,E2 -14537.286} C_VEL
LIN {X 0,Y 334.182,Z 636.164,A -85,B 0,C 180,E1 -14539.063,E2 -14539.063} C_VEL
LIN {X 0,Y 324.551,Z 655.099,A -85,B 0,C 180,E1 -14541.29,E2 -14541.29} C_VEL
LIN {X 0,Y 315.626,Z 672.769,A -85,B 0,C 180,E1 -14543.899,E2 -14543.899} C_VEL
LIN {X 0,Y 307.533,Z 689.18,A -85,B 0,C 180,E1 -14546.894,E2 -14546.894} C_VEL
LIN {X 0,Y 300.683,Z 703.374,A -85,B 0,C 180,E1 -14550.08,E2 -14550.08} C_VEL
LIN {X 0,Y 294.685,Z 716.038,A -85,B 0,C 180,E1 -14553.611,E2 -14553.611} C_VEL
LIN {X 0,Y 289.864,Z 726.446,A -85,B 0,C 180,E1 -14557.274,E2 -14557.274} C_VEL
LIN {X 0,Y 286.166,Z 734.798,A -85,B 0,C 180,E1 -14561.039,E2 -14561.039} C_VEL
LIN {X 0,Y 283.507,Z 741.218,A -85,B 0,C 180,E1 -14564.872,E2 -14564.872} C_VEL
LIN {X 0,Y 281.765,Z 745.798,A -85,B 0,C 180,E1 -14568.746,E2 -14568.746} C_VEL
LIN {X 0,Y 280.773,Z 748.591,A -85,B 0,C 180,E1 -14572.635,E2 -14572.635} C_VEL
LIN {X 0,Y 280.337,Z 749.626,A -85,B 0,C 180,E1 -14576.32,E2 -14576.32} C_VEL
LIN {X 0,Y 280.187,Z 749.061,A -85,B 0,C 180,E1 -14580.001,E2 -14580.001} C_VEL
LIN {X 0,Y 280.169,Z 746.862,A -85,B 0,C 180,E1 -14583.684,E2 -14583.684} C_VEL
LIN {X 0,Y 280.357,Z 742.956,A -85,B 0,C 180,E1 -14587.377,E2 -14587.377} C_VEL
LIN {X 0,Y 280.912,Z 737.225,A -85,B 0,C 180,E1 -14591.082,E2 -14591.082} C_VEL
LIN {X 0,Y 281.983,Z 729.517,A -85,B 0,C 180,E1 -14594.792,E2 -14594.792} C_VEL
LIN {X 0,Y 283.611,Z 720.236,A -85,B 0,C 180,E1 -14598.287,E2 -14598.287} C_VEL
LIN {X 0,Y 285.77,Z 709.469,A -85,B 0,C 180,E1 -14601.555,E2 -14601.555} C_VEL
LIN {X 0,Y 288.393,Z 697.285,A -85,B 0,C 180,E1 -14604.586,E2 -14604.586} C_VEL
LIN {X 0,Y 291.504,Z 683.172,A -85,B 0,C 180,E1 -14607.474,E2 -14607.474} C_VEL
LIN {X 0,Y 294.929,Z 667.46,A -85,B 0,C 180,E1 -14610.116,E2 -14610.116} C_VEL
LIN {X 0,Y 298.561,Z 650.003,A -85,B 0,C 180,E1 -14612.515,E2 -14612.515} C_VEL
LIN {X 0,Y 301.977,Z 632.326,A -85,B 0,C 180,E1 -14614.486,E2 -14614.486} C_VEL
LIN {X 0,Y 305.283,Z 613.192,A -85,B 0,C 180,E1 -14616.201,E2 -14616.201} C_VEL
LIN {X 0,Y 308.319,Z 592.759,A -85,B 0,C 180,E1 -14617.625,E2 -14617.625} C_VEL
LIN {X 0,Y 310.864,Z 571.524,A -85,B 0,C 180,E1 -14618.712,E2 -14618.712} C_VEL
LIN {X 0,Y 312.978,Z 547.09,A -85,B 0,C 180,E1 -14619.572,E2 -14619.572} C_VEL
LIN {X 0,Y 325.336,Z 390.045,A -85,B 0,C 180,E1 -14624.313,E2 -14624.313} C_VEL
LIN {X 0,Y 324.759,Z 387.177,A -85,B 0,C 180,E1 -14624.509,E2 -14624.509} C_VEL
LIN {X 0,Y 311.766,Z 362.38,A -85,B 0,C 180,E1 -14627.443,E2 -14627.443} C_VEL
LIN {X 0,Y 299.503,Z 340.601,A -85,B 0,C 180,E1 -14630.444,E2 -14630.444} C_VEL
LIN {X 0,Y 297.465,Z 336.802,A -85,B 0,C 180,E1 -14631.054,E2 -14631.054} C_VEL
LIN {X 0,Y 290.856,Z 320.692,A -85,B 0,C 180,E1 -14635.246,E2 -14635.246} C_VEL
LIN {X 0,Y 287.28,Z 312.589,A -85,B 0,C 180,E1 -14637.625,E2 -14637.625} C_VEL
LIN {X 0,Y 287.974,Z 312.566,A -85,B 0,C 180,E1 -14638.049,E2 -14638.049} C_VEL
LIN {X 0,Y 291.896,Z 320.133,A -85,B 0,C 180,E1 -14639.991,E2 -14639.991} C_VEL
LIN {X 0,Y 298.485,Z 334.191,A -85,B 0,C 180,E1 -14643.219,E2 -14643.219} C_VEL
LIN {X 0,Y 304.835,Z 349.874,A -85,B 0,C 180,E1 -14646.41,E2 -14646.41} C_VEL
LIN {X 0,Y 310.826,Z 367.12,A -85,B 0,C 180,E1 -14649.561,E2 -14649.561} C_VEL
LIN {X 0,Y 312.652,Z 373.507,A -85,B 0,C 180,E1 -14650.634,E2 -14650.634} C_VEL
LIN {X 0,Y 308.169,Z 414.628,A -85,B 0,C 180,E1 -14655.05,E2 -14655.05} C_VEL
LIN {X 0,Y 303.645,Z 457.497,A -85,B 0,C 180,E1 -14659.66,E2 -14659.66} C_VEL
LIN {X 0,Y 301.084,Z 483.752,A -85,B 0,C 180,E1 -14662.461,E2 -14662.461} C_VEL
LIN {X 0,Y 303.108,Z 507.473,A -85,B 0,C 180,E1 -14663.348,E2 -14663.348} C_VEL
LIN {X 0,Y 298.757,Z 627.929,A -85,B 0,C 180,E1 -14666.274,E2 -14666.274} C_VEL
LIN {X 0,Y 297.652,Z 644.202,A -85,B 0,C 180,E1 -14667.025,E2 -14667.025} C_VEL
LIN {X 0,Y 296.117,Z 659.427,A -85,B 0,C 180,E1 -14668.063,E2 -14668.063} C_VEL
LIN {X 0,Y 294.181,Z 673.985,A -85,B 0,C 180,E1 -14669.414,E2 -14669.414} C_VEL
LIN {X 0,Y 291.849,Z 688.476,A -85,B 0,C 180,E1 -14671.176,E2 -14671.176} C_VEL
LIN {X 0,Y 289.491,Z 701.221,A -85,B 0,C 180,E1 -14673.166,E2 -14673.166} C_VEL
LIN {X 0,Y 287.056,Z 713.46,A -85,B 0,C 180,E1 -14675.595,E2 -14675.595} C_VEL
LIN {X 0,Y 284.89,Z 723.782,A -85,B 0,C 180,E1 -14678.217,E2 -14678.217} C_VEL
LIN {X 0,Y 283.121,Z 732.348,A -85,B 0,C 180,E1 -14680.991,E2 -14680.991} C_VEL
LIN {X 0,Y 282.245,Z 736.774,A -85,B 0,C 180,E1 -14682.77,E2 -14682.77} C_VEL
LIN {X 0,Y 280.683,Z 739.906,A -85,B 0,C 180,E1 -14684.187,E2 -14684.187} C_VEL
LIN {X 0,Y 275.672,Z 744.607,A -85,B 0,C 180,E1 -14686.699,E2 -14686.699} C_VEL
LIN {X 0,Y 272.862,Z 747.256,A -85,B 0,C 180,E1 -14688.64,E2 -14688.64} C_VEL
LIN {X 0,Y 272.485,Z 748.065,A -85,B 0,C 180,E1 -14689.435,E2 -14689.435} C_VEL
LIN {X 0,Y 272.241,Z 750.478,A -85,B 0,C 180,E1 -14692.8,E2 -14692.8} C_VEL
LIN {X 0,Y 272.224,Z 751.109,A -85,B 0,C 180,E1 -14696.149,E2 -14696.149} C_VEL
LIN {X 0,Y 272.432,Z 750.061,A -85,B 0,C 180,E1 -14699.561,E2 -14699.561} C_VEL
LIN {X 0,Y 272.961,Z 747.379,A -85,B 0,C 180,E1 -14702.825,E2 -14702.825} C_VEL
LIN {X 0,Y 274.037,Z 742.664,A -85,B 0,C 180,E1 -14706.258,E2 -14706.258} C_VEL
LIN {X 0,Y 275.619,Z 736.449,A -85,B 0,C 180,E1 -14709.405,E2 -14709.405} C_VEL
LIN {X 0,Y 277.861,Z 727.994,A -85,B 0,C 180,E1 -14712.567,E2 -14712.567} C_VEL
LIN {X 0,Y 280.299,Z 718.761,A -85,B 0,C 180,E1 -14715.219,E2 -14715.219} C_VEL
LIN {X 0,Y 283.233,Z 707.063,A -85,B 0,C 180,E1 -14717.841,E2 -14717.841} C_VEL
LIN {X 0,Y 286.023,Z 694.923,A -85,B 0,C 180,E1 -14719.967,E2 -14719.967} C_VEL
LIN {X 0,Y 288.739,Z 681.488,A -85,B 0,C 180,E1 -14721.815,E2 -14721.815} C_VEL
LIN {X 0,Y 291.143,Z 667.519,A -85,B 0,C 180,E1 -14723.304,E2 -14723.304} C_VEL
LIN {X 0,Y 293.284,Z 651.386,A -85,B 0,C 180,E1 -14724.579,E2 -14724.579} C_VEL
LIN {X 0,Y 294.752,Z 635.543,A -85,B 0,C 180,E1 -14725.449,E2 -14725.449} C_VEL
LIN {X 0,Y 295.692,Z 617.171,A -85,B 0,C 180,E1 -14726.049,E2 -14726.049} C_VEL
LIN {X 0,Y 300.247,Z 506.37,A -85,B 0,C 180,E1 -14728.791,E2 -14728.791} C_VEL
LIN {X 0,Y 298.26,Z 484.586,A -85,B 0,C 180,E1 -14729.811,E2 -14729.811} C_VEL
LIN {X 0,Y 303.278,Z 441.118,A -85,B 0,C 180,E1 -14734.517,E2 -14734.517} C_VEL
LIN {X 0,Y 308.284,Z 400.374,A -85,B 0,C 180,E1 -14738.899,E2 -14738.899} C_VEL
LIN {X 0,Y 310.833,Z 378.715,A -85,B 0,C 180,E1 -14741.235,E2 -14741.235} C_VEL
LIN {X 0,Y 306.761,Z 365.002,A -85,B 0,C 180,E1 -14743.915,E2 -14743.915} C_VEL
LIN {X 0,Y 302.148,Z 352.38,A -85,B 0,C 180,E1 -14746.8,E2 -14746.8} C_VEL
LIN {X 0,Y 297.407,Z 341.469,A -85,B 0,C 180,E1 -14749.735,E2 -14749.735} C_VEL
LIN {X 0,Y 292.716,Z 332.185,A -85,B 0,C 180,E1 -14752.739,E2 -14752.739} C_VEL
LIN {X 0,Y 290.789,Z 328.5,A -85,B 0,C 180,E1 -14754.079,E2 -14754.079} C_VEL
LIN {X 0,Y 288.17,Z 324.01,A -85,B 0,C 180,E1 -14755.821,E2 -14755.821} C_VEL
LIN {X 0,Y 285.709,Z 319.489,A -85,B 0,C 180,E1 -14757.793,E2 -14757.793} C_VEL
LIN {X 0,Y 283.292,Z 316.154,A -85,B 0,C 180,E1 -14759.595,E2 -14759.595} C_VEL
LIN {X 0,Y 282.211,Z 313.989,A -85,B 0,C 180,E1 -14760.608,E2 -14760.608} C_VEL
LIN {X 0,Y 279.643,Z 310.853,A -85,B 0,C 180,E1 -14762.869,E2 -14762.869} C_VEL
LIN {X 0,Y 278.473,Z 308.311,A -85,B 0,C 180,E1 -14764.324,E2 -14764.324} C_VEL
LIN {X 0,Y 275.202,Z 304.808,A -85,B 0,C 180,E1 -14768.145,E2 -14768.145} C_VEL
LIN {X 0,Y 274.529,Z 302.767,A -85,B 0,C 180,E1 -14770.067,E2 -14770.067} C_VEL
LIN {X 0,Y 274.475,Z 302.286,A -85,B 0,C 180,E1 -14773.052,E2 -14773.052} C_VEL
LIN {X 0,Y 274.458,Z 302.294,A -85,B 0,C 180,E1 -14777.819,E2 -14777.819} C_VEL
LIN {X 0,Y 274.484,Z 302.316,A -85,B 0,C 180,E1 -14782.713,E2 -14782.713} C_VEL
LIN {X 0,Y 274.51,Z 302.633,A -85,B 0,C 180,E1 -14783.777,E2 -14783.777} C_VEL
LIN {X 0,Y 276.194,Z 306.361,A -85,B 0,C 180,E1 -14785.059,E2 -14785.059} C_VEL
LIN {X 0,Y 282.302,Z 319.458,A -85,B 0,C 180,E1 -14789.027,E2 -14789.027} C_VEL
LIN {X 0,Y 284.199,Z 323.388,A -85,B 0,C 180,E1 -14790.059,E2 -14790.059} C_VEL
LIN {X 0,Y 297.646,Z 344.923,A -85,B 0,C 180,E1 -14793.718,E2 -14793.718} C_VEL
LIN {X 0,Y 311.043,Z 367.574,A -85,B 0,C 180,E1 -14797.007,E2 -14797.007} C_VEL
LIN {X 0,Y 324.168,Z 391.398,A -85,B 0,C 180,E1 -14799.952,E2 -14799.952} C_VEL
LIN {X 0,Y 309.274,Z 576.305,A -85,B 0,C 180,E1 -14805.427,E2 -14805.427} C_VEL
LIN {X 0,Y 306.783,Z 597.161,A -85,B 0,C 180,E1 -14806.347,E2 -14806.347} C_VEL
LIN {X 0,Y 303.743,Z 617.505,A -85,B 0,C 180,E1 -14807.564,E2 -14807.564} C_VEL
LIN {X 0,Y 300.178,Z 637.626,A -85,B 0,C 180,E1 -14809.122,E2 -14809.122} C_VEL
LIN {X 0,Y 296.114,Z 657.791,A -85,B 0,C 180,E1 -14811.097,E2 -14811.097} C_VEL
LIN {X 0,Y 292.057,Z 676.129,A -85,B 0,C 180,E1 -14813.322,E2 -14813.322} C_VEL
LIN {X 0,Y 287.979,Z 693.486,A -85,B 0,C 180,E1 -14815.897,E2 -14815.897} C_VEL
LIN {X 0,Y 284.014,Z 709.769,A -85,B 0,C 180,E1 -14818.838,E2 -14818.838} C_VEL
LIN {X 0,Y 280.583,Z 723.971,A -85,B 0,C 180,E1 -14821.944,E2 -14821.944} C_VEL
LIN {X 0,Y 277.481,Z 737.412,A -85,B 0,C 180,E1 -14825.522,E2 -14825.522} C_VEL
LIN {X 0,Y 275.182,Z 748.503,A -85,B 0,C 180,E1 -14829.143,E2 -14829.143} C_VEL
LIN {X 0,Y 273.543,Z 758.012,A -85,B 0,C 180,E1 -14833,E2 -14833} C_VEL
LIN {X 0,Y 272.604,Z 765.487,A -85,B 0,C 180,E1 -14836.858,E2 -14836.858} C_VEL
LIN {X 0,Y 272.197,Z 772.186,A -85,B 0,C 180,E1 -14841.34,E2 -14841.34} C_VEL
LIN {X 0,Y 272.163,Z 775.703,A -85,B 0,C 180,E1 -14844.733,E2 -14844.733} C_VEL
LIN {X 0,Y 272.215,Z 777.363,A -85,B 0,C 180,E1 -14847.897,E2 -14847.897} C_VEL
LIN {X 0,Y 272.188,Z 777.946,A -85,B 0,C 180,E1 -14851.897,E2 -14851.897} C_VEL
LIN {X 0,Y 272.08,Z 777.126,A -85,B 0,C 180,E1 -14855.697,E2 -14855.697} C_VEL
LIN {X 0,Y 272.127,Z 774.839,A -85,B 0,C 180,E1 -14859.519,E2 -14859.519} C_VEL
LIN {X 0,Y 272.675,Z 770.631,A -85,B 0,C 180,E1 -14863.662,E2 -14863.662} C_VEL
LIN {X 0,Y 274.046,Z 764.625,A -85,B 0,C 180,E1 -14867.849,E2 -14867.849} C_VEL
LIN {X 0,Y 276.479,Z 756.619,A -85,B 0,C 180,E1 -14872.095,E2 -14872.095} C_VEL
LIN {X 0,Y 280.129,Z 746.625,A -85,B 0,C 180,E1 -14876.271,E2 -14876.271} C_VEL
LIN {X 0,Y 285.114,Z 734.504,A -85,B 0,C 180,E1 -14880.333,E2 -14880.333} C_VEL
LIN {X 0,Y 291.544,Z 720.009,A -85,B 0,C 180,E1 -14884.258,E2 -14884.258} C_VEL
LIN {X 0,Y 298.948,Z 704.206,A -85,B 0,C 180,E1 -14887.741,E2 -14887.741} C_VEL
LIN {X 0,Y 307.58,Z 686.563,A -85,B 0,C 180,E1 -14890.923,E2 -14890.923} C_VEL
LIN {X 0,Y 317.689,Z 666.722,A -85,B 0,C 180,E1 -14893.823,E2 -14893.823} C_VEL
LIN {X 0,Y 328.403,Z 646.394,A -85,B 0,C 180,E1 -14896.186,E2 -14896.186} C_VEL
LIN {X 0,Y 334.839,Z 634.376,A -85,B 0,C 180,E1 -14897.352,E2 -14897.352} C_VEL
LIN {X 0,Y 323.905,Z 653.14,A -85,B 0,C 180,E1 -14899.475,E2 -14899.475} C_VEL
LIN {X 0,Y 313.697,Z 670.924,A -85,B 0,C 180,E1 -14902.037,E2 -14902.037} C_VEL
LIN {X 0,Y 304.158,Z 687.883,A -85,B 0,C 180,E1 -14905.112,E2 -14905.112} C_VEL
LIN {X 0,Y 296.096,Z 702.657,A -85,B 0,C 180,E1 -14908.44,E2 -14908.44} C_VEL
LIN {X 0,Y 289.375,Z 715.279,A -85,B 0,C 180,E1 -14911.972,E2 -14911.972} C_VEL
LIN {X 0,Y 283.92,Z 725.821,A -85,B 0,C 180,E1 -14915.668,E2 -14915.668} C_VEL
LIN {X 0,Y 279.598,Z 734.456,A -85,B 0,C 180,E1 -14919.546,E2 -14919.546} C_VEL
LIN {X 0,Y 276.353,Z 741.257,A -85,B 0,C 180,E1 -14923.609,E2 -14923.609} C_VEL
LIN {X 0,Y 274.263,Z 745.975,A -85,B 0,C 180,E1 -14927.58,E2 -14927.58} C_VEL
LIN {X 0,Y 273.02,Z 748.937,A -85,B 0,C 180,E1 -14931.577,E2 -14931.577} C_VEL
LIN {X 0,Y 272.416,Z 750.157,A -85,B 0,C 180,E1 -14935.58,E2 -14935.58} C_VEL
LIN {X 0,Y 272.211,Z 749.687,A -85,B 0,C 180,E1 -14939.369,E2 -14939.369} C_VEL
LIN {X 0,Y 272.167,Z 747.573,A -85,B 0,C 180,E1 -14943.16,E2 -14943.16} C_VEL
LIN {X 0,Y 272.307,Z 744.018,A -85,B 0,C 180,E1 -14946.749,E2 -14946.749} C_VEL
LIN {X 0,Y 272.76,Z 738.867,A -85,B 0,C 180,E1 -14950.348,E2 -14950.348} C_VEL
LIN {X 0,Y 273.669,Z 731.999,A -85,B 0,C 180,E1 -14953.954,E2 -14953.954} C_VEL
LIN {X 0,Y 275.176,Z 723.231,A -85,B 0,C 180,E1 -14957.554,E2 -14957.554} C_VEL
LIN {X 0,Y 277.223,Z 713.013,A -85,B 0,C 180,E1 -14960.921,E2 -14960.921} C_VEL
LIN {X 0,Y 279.753,Z 701.429,A -85,B 0,C 180,E1 -14964.045,E2 -14964.045} C_VEL
LIN {X 0,Y 282.902,Z 687.553,A -85,B 0,C 180,E1 -14967.125,E2 -14967.125} C_VEL
LIN {X 0,Y 286.29,Z 672.63,A -85,B 0,C 180,E1 -14969.847,E2 -14969.847} C_VEL
LIN {X 0,Y 289.906,Z 656.104,A -85,B 0,C 180,E1 -14972.327,E2 -14972.327} C_VEL
LIN {X 0,Y 293.625,Z 637.936,A -85,B 0,C 180,E1 -14974.54,E2 -14974.54} C_VEL
LIN {X 0,Y 297.011,Z 619.609,A -85,B 0,C 180,E1 -14976.335,E2 -14976.335} C_VEL
LIN {X 0,Y 300.092,Z 600.611,A -85,B 0,C 180,E1 -14977.812,E2 -14977.812} C_VEL
LIN {X 0,Y 302.879,Z 580.053,A -85,B 0,C 180,E1 -14979.033,E2 -14979.033} C_VEL
LIN {X 0,Y 305.192,Z 558.06,A -85,B 0,C 180,E1 -14979.959,E2 -14979.959} C_VEL
LIN {X 0,Y 318.928,Z 391.443,A -85,B 0,C 180,E1 -14985.137,E2 -14985.137} C_VEL
LIN {X 0,Y 306.393,Z 367.361,A -85,B 0,C 180,E1 -14988.041,E2 -14988.041} C_VEL
LIN {X 0,Y 294.454,Z 345.957,A -85,B 0,C 180,E1 -14991.05,E2 -14991.05} C_VEL
LIN {X 0,Y 289.228,Z 336.759,A -85,B 0,C 180,E1 -14992.522,E2 -14992.522} C_VEL
LIN {X 0,Y 283.078,Z 321.912,A -85,B 0,C 180,E1 -14996.562,E2 -14996.562} C_VEL
LIN {X 0,Y 281.913,Z 319.289,A -85,B 0,C 180,E1 -14997.376,E2 -14997.376} C_VEL
LIN {X 0,Y 282.497,Z 319.09,A -85,B 0,C 180,E1 -14997.771,E2 -14997.771} C_VEL
LIN {X 0,Y 283.327,Z 319.53,A -85,B 0,C 180,E1 -14998.036,E2 -14998.036} C_VEL
LIN {X 0,Y 288.214,Z 329.516,A -85,B 0,C 180,E1 -15000.548,E2 -15000.548} C_VEL
LIN {X 0,Y 294.105,Z 342.745,A -85,B 0,C 180,E1 -15003.552,E2 -15003.552} C_VEL
LIN {X 0,Y 300.291,Z 358.685,A -85,B 0,C 180,E1 -15006.779,E2 -15006.779} C_VEL
LIN {X 0,Y 305.477,Z 374.744,A -85,B 0,C 180,E1 -15009.697,E2 -15009.697} C_VEL
LIN {X 0,Y 305.898,Z 376.841,A -85,B 0,C 180,E1 -15010.026,E2 -15010.026} C_VEL
LIN {X 0,Y 301.217,Z 418.061,A -85,B 0,C 180,E1 -15014.5,E2 -15014.5} C_VEL
LIN {X 0,Y 296.144,Z 463.899,A -85,B 0,C 180,E1 -15019.493,E2 -15019.493} C_VEL
LIN {X 0,Y 294.131,Z 483.973,A -85,B 0,C 180,E1 -15021.667,E2 -15021.667} C_VEL
LIN {X 0,Y 296.154,Z 508.29,A -85,B 0,C 180,E1 -15022.6,E2 -15022.6} C_VEL
LIN {X 0,Y 291.612,Z 628.311,A -85,B 0,C 180,E1 -15025.58,E2 -15025.58} C_VEL
LIN {X 0,Y 290.461,Z 644.577,A -85,B 0,C 180,E1 -15026.347,E2 -15026.347} C_VEL
LIN {X 0,Y 288.844,Z 659.963,A -85,B 0,C 180,E1 -15027.419,E2 -15027.419} C_VEL
LIN {X 0,Y 286.828,Z 674.479,A -85,B 0,C 180,E1 -15028.799,E2 -15028.799} C_VEL
LIN {X 0,Y 284.4,Z 688.956,A -85,B 0,C 180,E1 -15030.602,E2 -15030.602} C_VEL
LIN {X 0,Y 281.941,Z 701.682,A -85,B 0,C 180,E1 -15032.64,E2 -15032.64} C_VEL
LIN {X 0,Y 279.398,Z 713.914,A -85,B 0,C 180,E1 -15035.131,E2 -15035.131} C_VEL
LIN {X 0,Y 277.25,Z 723.696,A -85,B 0,C 180,E1 -15037.666,E2 -15037.666} C_VEL
LIN {X 0,Y 275.277,Z 732.784,A -85,B 0,C 180,E1 -15040.673,E2 -15040.673} C_VEL
LIN {X 0,Y 273.835,Z 739.852,A -85,B 0,C 180,E1 -15043.768,E2 -15043.768} C_VEL
LIN {X 0,Y 272.879,Z 745.29,A -85,B 0,C 180,E1 -15047.043,E2 -15047.043} C_VEL
LIN {X 0,Y 272.485,Z 748.065,A -85,B 0,C 180,E1 -15049.435,E2 -15049.435} C_VEL
LIN {X 0,Y 271.339,Z 749.481,A -85,B 0,C 180,E1 -15051.025,E2 -15051.025} C_VEL
LIN {X 0,Y 267.308,Z 751.012,A -85,B 0,C 180,E1 -15053.609,E2 -15053.609} C_VEL
LIN {X 0,Y 264.503,Z 751.52,A -85,B 0,C 180,E1 -15055.951,E2 -15055.951} C_VEL
LIN {X 0,Y 264.253,Z 751.461,A -85,B 0,C 180,E1 -15056.799,E2 -15056.799} C_VEL
LIN {X 0,Y 264.517,Z 750.226,A -85,B 0,C 180,E1 -15060.178,E2 -15060.178} C_VEL
LIN {X 0,Y 265.178,Z 747.189,A -85,B 0,C 180,E1 -15063.657,E2 -15063.657} C_VEL
LIN {X 0,Y 266.324,Z 742.674,A -85,B 0,C 180,E1 -15066.916,E2 -15066.916} C_VEL
LIN {X 0,Y 268.09,Z 736.211,A -85,B 0,C 180,E1 -15070.178,E2 -15070.178} C_VEL
LIN {X 0,Y 270.38,Z 728.136,A -85,B 0,C 180,E1 -15073.238,E2 -15073.238} C_VEL
LIN {X 0,Y 273.042,Z 718.578,A -85,B 0,C 180,E1 -15076.015,E2 -15076.015} C_VEL
LIN {X 0,Y 276.104,Z 707.026,A -85,B 0,C 180,E1 -15078.643,E2 -15078.643} C_VEL
LIN {X 0,Y 278.939,Z 695.288,A -85,B 0,C 180,E1 -15080.733,E2 -15080.733} C_VEL
LIN {X 0,Y 281.852,Z 681.584,A -85,B 0,C 180,E1 -15082.654,E2 -15082.654} C_VEL
LIN {X 0,Y 284.332,Z 667.76,A -85,B 0,C 180,E1 -15084.147,E2 -15084.147} C_VEL
LIN {X 0,Y 286.547,Z 651.795,A -85,B 0,C 180,E1 -15085.43,E2 -15085.43} C_VEL
LIN {X 0,Y 288.086,Z 635.941,A -85,B 0,C 180,E1 -15086.315,E2 -15086.315} C_VEL
LIN {X 0,Y 289.074,Z 617.515,A -85,B 0,C 180,E1 -15086.927,E2 -15086.927} C_VEL
LIN {X 0,Y 293.842,Z 507.243,A -85,B 0,C 180,E1 -15089.711,E2 -15089.711} C_VEL
LIN {X 0,Y 291.897,Z 484.925,A -85,B 0,C 180,E1 -15090.793,E2 -15090.793} C_VEL
LIN {X 0,Y 297.347,Z 440.426,A -85,B 0,C 180,E1 -15095.674,E2 -15095.674} C_VEL
LIN {X 0,Y 302.688,Z 399.075,A -85,B 0,C 180,E1 -15100.171,E2 -15100.171} C_VEL
LIN {X 0,Y 304.731,Z 382.077,A -85,B 0,C 180,E1 -15102.035,E2 -15102.035} C_VEL
LIN {X 0,Y 300.846,Z 368.621,A -85,B 0,C 180,E1 -15104.777,E2 -15104.777} C_VEL
LIN {X 0,Y 296.367,Z 356.318,A -85,B 0,C 180,E1 -15107.728,E2 -15107.728} C_VEL
LIN {X 0,Y 292.051,Z 346.383,A -85,B 0,C 180,E1 -15110.541,E2 -15110.541} C_VEL
LIN {X 0,Y 288.167,Z 338.303,A -85,B 0,C 180,E1 -15113.224,E2 -15113.224} C_VEL
LIN {X 0,Y 285.708,Z 333.699,A -85,B 0,C 180,E1 -15114.98,E2 -15114.98} C_VEL
LIN {X 0,Y 284.125,Z 330.703,A -85,B 0,C 180,E1 -15116.165,E2 -15116.165} C_VEL
LIN {X 0,Y 281.48,Z 325.966,A -85,B 0,C 180,E1 -15118.371,E2 -15118.371} C_VEL
LIN {X 0,Y 279.059,Z 321.939,A -85,B 0,C 180,E1 -15120.41,E2 -15120.41} C_VEL
LIN {X 0,Y 278.421,Z 320.879,A -85,B 0,C 180,E1 -15121.028,E2 -15121.028} C_VEL
LIN {X 0,Y 276.082,Z 317.675,A -85,B 0,C 180,E1 -15123.321,E2 -15123.321} C_VEL
LIN {X 0,Y 275.114,Z 315.512,A -85,B 0,C 180,E1 -15124.585,E2 -15124.585} C_VEL
LIN {X 0,Y 272.087,Z 312.03,A -85,B 0,C 180,E1 -15128.452,E2 -15128.452} C_VEL
LIN {X 0,Y 271.128,Z 309.776,A -85,B 0,C 180,E1 -15130.625,E2 -15130.625} C_VEL
LIN {X 0,Y 269.324,Z 308.419,A -85,B 0,C 180,E1 -15136.388,E2 -15136.388} C_VEL
LIN {X 0,Y 270.346,Z 309.154,A -85,B 0,C 180,E1 -15142.398,E2 -15142.398} C_VEL
LIN {X 0,Y 270.762,Z 309.633,A -85,B 0,C 180,E1 -15143.388,E2 -15143.388} C_VEL
LIN {X 0,Y 271.139,Z 313.626,A -85,B 0,C 180,E1 -15145.325,E2 -15145.325} C_VEL
LIN {X 0,Y 275.742,Z 323.281,A -85,B 0,C 180,E1 -15148.301,E2 -15148.301} C_VEL
LIN {X 0,Y 287.772,Z 342.313,A -85,B 0,C 180,E1 -15151.79,E2 -15151.79} C_VEL
LIN {X 0,Y 301.06,Z 364.388,A -85,B 0,C 180,E1 -15155.242,E2 -15155.242} C_VEL
LIN {X 0,Y 315.589,Z 390.323,A -85,B 0,C 180,E1 -15158.677,E2 -15158.677} C_VEL
LIN {X 0,Y 317.619,Z 394.628,A -85,B 0,C 180,E1 -15159.155,E2 -15159.155} C_VEL
LIN {X 0,Y 302.389,Z 575.956,A -85,B 0,C 180,E1 -15164.662,E2 -15164.662} C_VEL
LIN {X 0,Y 299.775,Z 597.094,A -85,B 0,C 180,E1 -15165.617,E2 -15165.617} C_VEL
LIN {X 0,Y 296.47,Z 618.357,A -85,B 0,C 180,E1 -15166.93,E2 -15166.93} C_VEL
LIN {X 0,Y 292.818,Z 638.227,A -85,B 0,C 180,E1 -15168.518,E2 -15168.518} C_VEL
LIN {X 0,Y 288.629,Z 658.3,A -85,B 0,C 180,E1 -15170.546,E2 -15170.546} C_VEL
LIN {X 0,Y 284.486,Z 676.419,A -85,B 0,C 180,E1 -15172.809,E2 -15172.809} C_VEL
LIN {X 0,Y 280.294,Z 693.704,A -85,B 0,C 180,E1 -15175.449,E2 -15175.449} C_VEL
LIN {X 0,Y 276.223,Z 709.913,A -85,B 0,C 180,E1 -15178.466,E2 -15178.466} C_VEL
LIN {X 0,Y 272.596,Z 724.476,A -85,B 0,C 180,E1 -15181.763,E2 -15181.763} C_VEL
LIN {X 0,Y 269.51,Z 737.495,A -85,B 0,C 180,E1 -15185.356,E2 -15185.356} C_VEL
LIN {X 0,Y 267.122,Z 748.76,A -85,B 0,C 180,E1 -15189.173,E2 -15189.173} C_VEL
LIN {X 0,Y 265.488,Z 758.169,A -85,B 0,C 180,E1 -15193.145,E2 -15193.145} C_VEL
LIN {X 0,Y 264.401,Z 767.852,A -85,B 0,C 180,E1 -15198.356,E2 -15198.356} C_VEL
LIN {X 0,Y 264.19,Z 772.658,A -85,B 0,C 180,E1 -15201.734,E2 -15201.734} C_VEL
LIN {X 0,Y 264.168,Z 775.682,A -85,B 0,C 180,E1 -15205.008,E2 -15205.008} C_VEL
LIN {X 0,Y 264.23,Z 777.064,A -85,B 0,C 180,E1 -15208.268,E2 -15208.268} C_VEL
LIN {X 0,Y 264.177,Z 777.43,A -85,B 0,C 180,E1 -15212.605,E2 -15212.605} C_VEL
LIN {X 0,Y 264.077,Z 776.453,A -85,B 0,C 180,E1 -15216.524,E2 -15216.524} C_VEL
LIN {X 0,Y 264.221,Z 773.841,A -85,B 0,C 180,E1 -15220.688,E2 -15220.688} C_VEL
LIN {X 0,Y 265.035,Z 769.328,A -85,B 0,C 180,E1 -15225.09,E2 -15225.09} C_VEL
LIN {X 0,Y 266.946,Z 762.598,A -85,B 0,C 180,E1 -15229.702,E2 -15229.702} C_VEL
LIN {X 0,Y 270.168,Z 753.796,A -85,B 0,C 180,E1 -15234.257,E2 -15234.257} C_VEL
LIN {X 0,Y 274.854,Z 742.845,A -85,B 0,C 180,E1 -15238.7,E2 -15238.7} C_VEL
LIN {X 0,Y 280.928,Z 729.973,A -85,B 0,C 180,E1 -15242.866,E2 -15242.866} C_VEL
LIN {X 0,Y 288.198,Z 715.598,A -85,B 0,C 180,E1 -15246.638,E2 -15246.638} C_VEL
LIN {X 0,Y 297.183,Z 698.695,A -85,B 0,C 180,E1 -15250.241,E2 -15250.241} C_VEL
LIN {X 0,Y 307.868,Z 679.659,A -85,B 0,C 180,E1 -15253.514,E2 -15253.514} C_VEL
LIN {X 0,Y 319.374,Z 660.145,A -85,B 0,C 180,E1 -15256.191,E2 -15256.191} C_VEL
LIN {X 0,Y 325.765,Z 649.611,A -85,B 0,C 180,E1 -15257.414,E2 -15257.414} C_VEL
LIN {X 0,Y 314.262,Z 666.991,A -85,B 0,C 180,E1 -15259.77,E2 -15259.77} C_VEL
LIN {X 0,Y 303.398,Z 683.845,A -85,B 0,C 180,E1 -15262.673,E2 -15262.673} C_VEL
LIN {X 0,Y 293.68,Z 699.52,A -85,B 0,C 180,E1 -15266.059,E2 -15266.059} C_VEL
LIN {X 0,Y 285.522,Z 712.972,A -85,B 0,C 180,E1 -15269.718,E2 -15269.718} C_VEL
LIN {X 0,Y 278.856,Z 724.281,A -85,B 0,C 180,E1 -15273.602,E2 -15273.602} C_VEL
LIN {X 0,Y 273.596,Z 733.507,A -85,B 0,C 180,E1 -15277.663,E2 -15277.663} C_VEL
LIN {X 0,Y 269.833,Z 740.386,A -85,B 0,C 180,E1 -15281.642,E2 -15281.642} C_VEL
LIN {X 0,Y 267.139,Z 745.587,A -85,B 0,C 180,E1 -15285.795,E2 -15285.795} C_VEL
LIN {X 0,Y 265.515,Z 748.851,A -85,B 0,C 180,E1 -15289.806,E2 -15289.806} C_VEL
LIN {X 0,Y 264.629,Z 750.502,A -85,B 0,C 180,E1 -15293.928,E2 -15293.928} C_VEL
LIN {X 0,Y 264.272,Z 750.466,A -85,B 0,C 180,E1 -15297.833,E2 -15297.833} C_VEL
LIN {X 0,Y 264.172,Z 748.978,A -85,B 0,C 180,E1 -15301.519,E2 -15301.519} C_VEL
LIN {X 0,Y 264.223,Z 746.024,A -85,B 0,C 180,E1 -15305.212,E2 -15305.212} C_VEL
LIN {X 0,Y 264.563,Z 741.161,A -85,B 0,C 180,E1 -15309.134,E2 -15309.134} C_VEL
LIN {X 0,Y 265.386,Z 734.396,A -85,B 0,C 180,E1 -15313.066,E2 -15313.066} C_VEL
LIN {X 0,Y 266.762,Z 726.114,A -85,B 0,C 180,E1 -15316.775,E2 -15316.775} C_VEL
LIN {X 0,Y 268.769,Z 716.047,A -85,B 0,C 180,E1 -15320.363,E2 -15320.363} C_VEL
LIN {X 0,Y 271.308,Z 704.577,A -85,B 0,C 180,E1 -15323.685,E2 -15323.685} C_VEL
LIN {X 0,Y 274.417,Z 691.206,A -85,B 0,C 180,E1 -15326.86,E2 -15326.86} C_VEL
LIN {X 0,Y 277.91,Z 676.283,A -85,B 0,C 180,E1 -15329.769,E2 -15329.769} C_VEL
LIN {X 0,Y 281.671,Z 659.728,A -85,B 0,C 180,E1 -15332.414,E2 -15332.414} C_VEL
LIN {X 0,Y 285.44,Z 642.18,A -85,B 0,C 180,E1 -15334.697,E2 -15334.697} C_VEL
LIN {X 0,Y 289.012,Z 623.955,A -85,B 0,C 180,E1 -15336.616,E2 -15336.616} C_VEL
LIN {X 0,Y 292.376,Z 604.552,A -85,B 0,C 180,E1 -15338.243,E2 -15338.243} C_VEL
LIN {X 0,Y 295.434,Z 583.617,A -85,B 0,C 180,E1 -15339.586,E2 -15339.586} C_VEL
LIN {X 0,Y 297.858,Z 562.33,A -85,B 0,C 180,E1 -15340.562,E2 -15340.562} C_VEL
LIN {X 0,Y 312.395,Z 394.234,A -85,B 0,C 180,E1 -15345.944,E2 -15345.944} C_VEL
LIN {X 0,Y 298.925,Z 368.327,A -85,B 0,C 180,E1 -15349.192,E2 -15349.192} C_VEL
LIN {X 0,Y 286.528,Z 346.299,A -85,B 0,C 180,E1 -15352.454,E2 -15352.454} C_VEL
LIN {X 0,Y 281.032,Z 336.77,A -85,B 0,C 180,E1 -15354.051,E2 -15354.051} C_VEL
LIN {X 0,Y 276.536,Z 325.965,A -85,B 0,C 180,E1 -15357.154,E2 -15357.154} C_VEL
LIN {X 0,Y 277.206,Z 325.934,A -85,B 0,C 180,E1 -15357.569,E2 -15357.569} C_VEL
LIN {X 0,Y 278.533,Z 326.078,A -85,B 0,C 180,E1 -15357.908,E2 -15357.908} C_VEL
LIN {X 0,Y 285.392,Z 340.857,A -85,B 0,C 180,E1 -15361.568,E2 -15361.568} C_VEL
LIN {X 0,Y 291.909,Z 357.019,A -85,B 0,C 180,E1 -15365.081,E2 -15365.081} C_VEL
LIN {X 0,Y 297.344,Z 372.904,A -85,B 0,C 180,E1 -15368.141,E2 -15368.141} C_VEL
LIN {X 0,Y 299.23,Z 379.812,A -85,B 0,C 180,E1 -15369.346,E2 -15369.346} C_VEL
LIN {X 0,Y 294.192,Z 422.409,A -85,B 0,C 180,E1 -15374.019,E2 -15374.019} C_VEL
LIN {X 0,Y 288.952,Z 467.762,A -85,B 0,C 180,E1 -15379.027,E2 -15379.027} C_VEL
LIN {X 0,Y 287.226,Z 484.319,A -85,B 0,C 180,E1 -15380.847,E2 -15380.847} C_VEL
LIN {X 0,Y 289.214,Z 509.1,A -85,B 0,C 180,E1 -15381.827,E2 -15381.827} C_VEL
LIN {X 0,Y 284.508,Z 628.629,A -85,B 0,C 180,E1 -15384.851,E2 -15384.851} C_VEL
LIN {X 0,Y 283.309,Z 644.913,A -85,B 0,C 180,E1 -15385.634,E2 -15385.634} C_VEL
LIN {X 0,Y 281.525,Z 661.149,A -85,B 0,C 180,E1 -15386.796,E2 -15386.796} C_VEL
LIN {X 0,Y 279.362,Z 675.851,A -85,B 0,C 180,E1 -15388.254,E2 -15388.254} C_VEL
LIN {X 0,Y 276.849,Z 690.156,A -85,B 0,C 180,E1 -15390.101,E2 -15390.101} C_VEL
LIN {X 0,Y 274.178,Z 703.264,A -85,B 0,C 180,E1 -15392.297,E2 -15392.297} C_VEL
LIN {X 0,Y 271.76,Z 714.369,A -85,B 0,C 180,E1 -15394.64,E2 -15394.64} C_VEL
LIN {X 0,Y 269.511,Z 724.138,A -85,B 0,C 180,E1 -15397.244,E2 -15397.244} C_VEL
LIN {X 0,Y 267.442,Z 733.22,A -85,B 0,C 180,E1 -15400.335,E2 -15400.335} C_VEL
LIN {X 0,Y 265.941,Z 740.196,A -85,B 0,C 180,E1 -15403.477,E2 -15403.477} C_VEL
LIN {X 0,Y 264.918,Z 745.708,A -85,B 0,C 180,E1 -15406.892,E2 -15406.892} C_VEL
LIN {X 0,Y 264.403,Z 749.31,A -85,B 0,C 180,E1 -15410.307,E2 -15410.307} C_VEL
LIN {X 0,Y 264.224,Z 751.237,A -85,B 0,C 180,E1 -15413.882,E2 -15413.882} C_VEL
LIN {X 0,Y 264.253,Z 751.461,A -85,B 0,C 180,E1 -15416.799,E2 -15416.799} C_VEL
LIN {X 0,Y 263.343,Z 751.16,A -85,B 0,C 180,E1 -15418.471,E2 -15418.471} C_VEL
LIN {X 0,Y 259.575,Z 749.852,A -85,B 0,C 180,E1 -15421.285,E2 -15421.285} C_VEL
LIN {X 0,Y 257.435,Z 748.046,A -85,B 0,C 180,E1 -15423.562,E2 -15423.562} C_VEL
LIN {X 0,Y 257.406,Z 747.146,A -85,B 0,C 180,E1 -15424.411,E2 -15424.411} C_VEL
LIN {X 0,Y 258.784,Z 742.152,A -85,B 0,C 180,E1 -15427.899,E2 -15427.899} C_VEL
LIN {X 0,Y 260.819,Z 735.313,A -85,B 0,C 180,E1 -15431.289,E2 -15431.289} C_VEL
LIN {X 0,Y 263.284,Z 727.137,A -85,B 0,C 180,E1 -15434.324,E2 -15434.324} C_VEL
LIN {X 0,Y 266.204,Z 717.225,A -85,B 0,C 180,E1 -15437.168,E2 -15437.168} C_VEL
LIN {X 0,Y 269.174,Z 706.501,A -85,B 0,C 180,E1 -15439.59,E2 -15439.59} C_VEL
LIN {X 0,Y 272.289,Z 694.083,A -85,B 0,C 180,E1 -15441.792,E2 -15441.792} C_VEL
LIN {X 0,Y 275.306,Z 680.345,A -85,B 0,C 180,E1 -15443.701,E2 -15443.701} C_VEL
LIN {X 0,Y 278.057,Z 665.111,A -85,B 0,C 180,E1 -15445.299,E2 -15445.299} C_VEL
LIN {X 0,Y 280.097,Z 650.585,A -85,B 0,C 180,E1 -15446.439,E2 -15446.439} C_VEL
LIN {X 0,Y 281.68,Z 634.015,A -85,B 0,C 180,E1 -15447.328,E2 -15447.328} C_VEL
LIN {X 0,Y 282.694,Z 614.703,A -85,B 0,C 180,E1 -15447.935,E2 -15447.935} C_VEL
LIN {X 0,Y 287.556,Z 508.326,A -85,B 0,C 180,E1 -15450.669,E2 -15450.669} C_VEL
LIN {X 0,Y 285.615,Z 485.555,A -85,B 0,C 180,E1 -15451.796,E2 -15451.796} C_VEL
LIN {X 0,Y 291.235,Z 441.939,A -85,B 0,C 180,E1 -15456.638,E2 -15456.638} C_VEL
